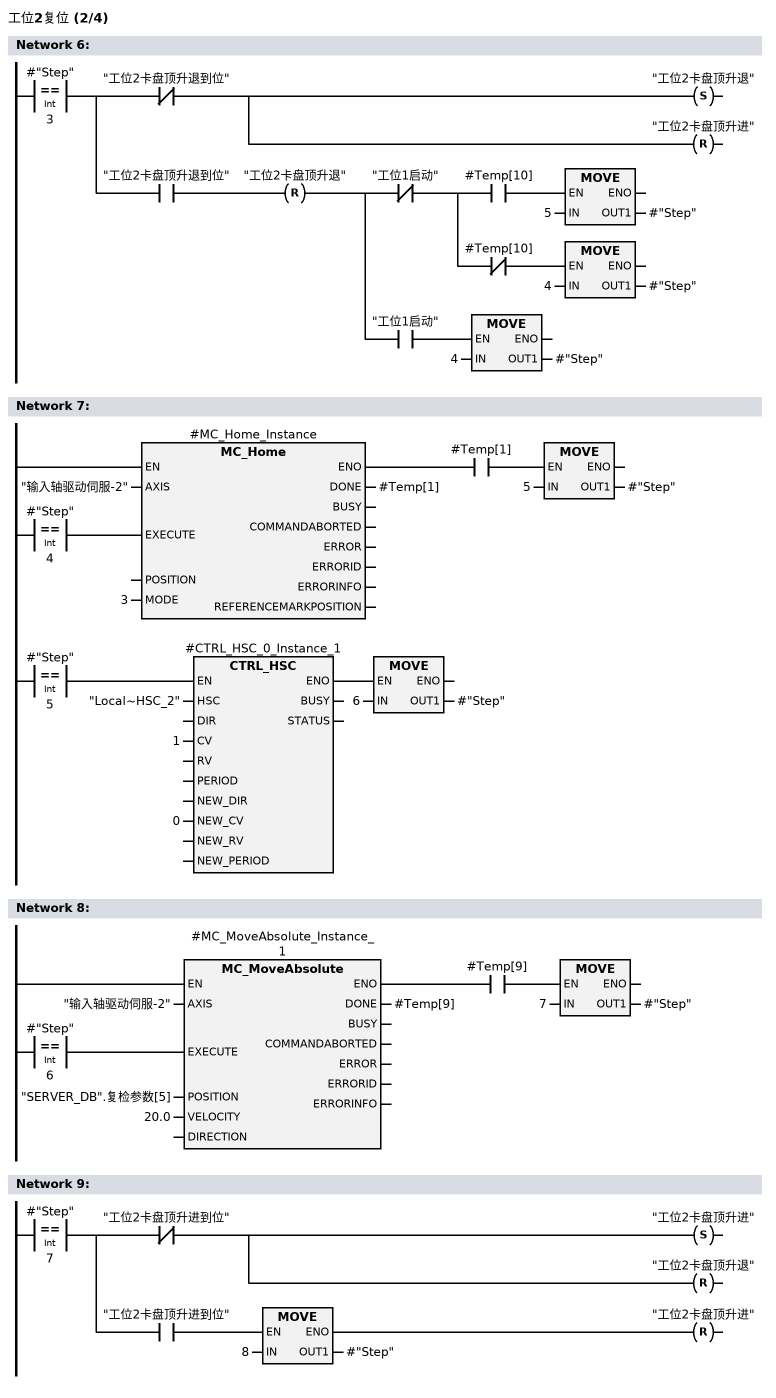
   RUNG wire#powerrail
      { S7_Templates := "SrcType := Int" } EQ_Contact(in1 := #"Step", in2 := 3)
      wire#w1
      I_Contact( "工位2卡盘顶升退到位" )
      wire#w2
      S_Coil( "工位2卡盘顶升退" )
   END_RUNG
   RUNG wire#w2
      R_Coil( "工位2卡盘顶升进" )
   END_RUNG
   RUNG wire#w1
      Contact( "工位2卡盘顶升退到位" )
      R_Coil( "工位2卡盘顶升退" )
      wire#w3
      I_Contact( "工位1启动" )
      wire#w4
      Contact( #Temp[10] )
      Move(in := 5, out1 => #"Step")
   END_RUNG
   RUNG wire#w4
      I_Contact( #Temp[10] )
      Move(in := 4, out1 => #"Step")
   END_RUNG
   RUNG wire#w3
      Contact( "工位1启动" )
      Move(in := 4, out1 => #"Step")
   END_RUNG
   // the same network as SCL:
   #_w1 := #"Step" = 3;
   IF #_w1 AND NOT "工位2卡盘顶升退到位" THEN
       "工位2卡盘顶升退" := TRUE;
       "工位2卡盘顶升进" := FALSE;
   END_IF;
   #_w2 := #_w1 AND "工位2卡盘顶升退到位";
   IF #_w2 THEN "工位2卡盘顶升退" := FALSE; END_IF;
   #_w3 := #_w2 AND NOT "工位1启动";
   IF #_w3 AND #Temp[10] THEN #"Step" := 5; END_IF;
   IF #_w3 AND NOT #Temp[10] THEN #"Step" := 4; END_IF;
   IF #_w2 AND "工位1启动" THEN #"Step" := 4; END_IF;
END_REGION

REGION Network 7
   // ENO of a box is taken as its EN; it also drops when the box reports an error
   #MC_Home_Instance(Axis := "输入轴驱动伺服-2", Execute := #"Step" = 4, Mode := 3, Done => #Temp[1]);   // MC_Home
   IF #Temp[1] THEN #"Step" := 5; END_IF;
   IF #"Step" = 5 THEN
       #CTRL_HSC_0_Instance_1(HSC := "Local~HSC_2", CV := 1, NEW_CV := 0);   // CTRL_HSC
       #"Step" := 6;
   END_IF;
END_REGION

REGION Network 8
   // ENO of a box is taken as its EN; it also drops when the box reports an error
   #MC_MoveAbsolute_Instance_1(Axis := "输入轴驱动伺服-2",   // MC_MoveAbsolute
                           Execute := #"Step" = 6,
                           Position := "SERVER_DB".复检参数[5],
                           Velocity := 20.0,
                           Done => #Temp[9]);
   IF #Temp[9] THEN #"Step" := 7; END_IF;
END_REGION

REGION Network 9
   RUNG wire#powerrail
      { S7_Templates := "SrcType := Int" } EQ_Contact(in1 := #"Step", in2 := 7)
      wire#w1
      I_Contact( "工位2卡盘顶升进到位" )
      wire#w2
      S_Coil( "工位2卡盘顶升进" )
   END_RUNG
   RUNG wire#w2
      R_Coil( "工位2卡盘顶升退" )
   END_RUNG
   RUNG wire#w1
      Contact( "工位2卡盘顶升进到位" )
      Move(in := 8, out1 => #"Step")
      R_Coil( "工位2卡盘顶升进" )
   END_RUNG
   // the same network as SCL:
   #_w1 := #"Step" = 7;
   IF #_w1 AND NOT "工位2卡盘顶升进到位" THEN
       "工位2卡盘顶升进" := TRUE;
       "工位2卡盘顶升退" := FALSE;
   END_IF;
   IF #_w1 AND "工位2卡盘顶升进到位" THEN
       #"Step" := 8;
       "工位2卡盘顶升进" := FALSE;
   END_IF;
END_REGION

REGION Network 10
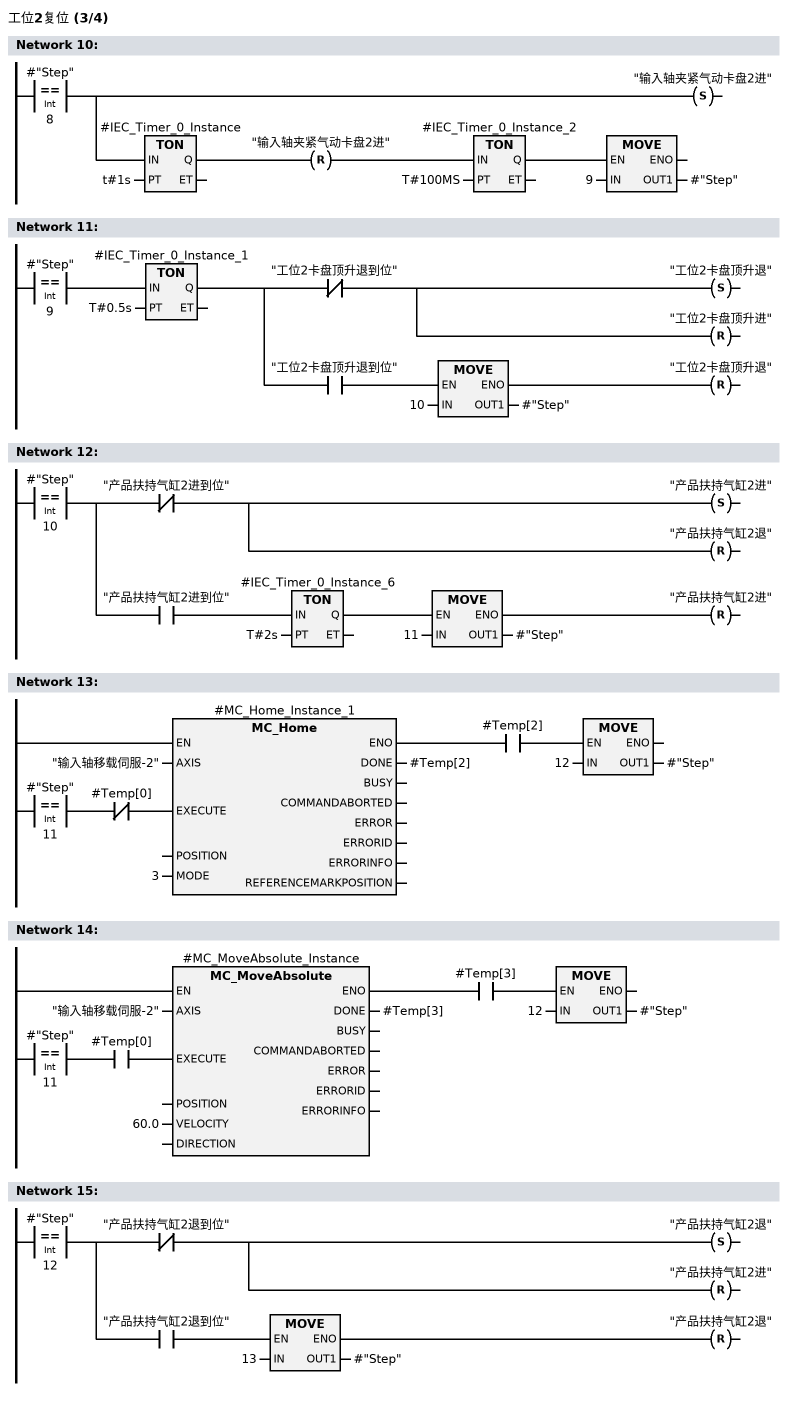
   #_w1 := #"Step" = 8;
   IF #_w1 THEN "输入轴夹紧气动卡盘2进" := TRUE; END_IF;
   #IEC_Timer_0_Instance(IN := #_w1, PT := t#1s);   // TON
   IF #IEC_Timer_0_Instance.Q THEN "输入轴夹紧气动卡盘2进" := FALSE; END_IF;
   #IEC_Timer_0_Instance_2(IN := #IEC_Timer_0_Instance.Q, PT := T#100MS);   // TON
   IF #IEC_Timer_0_Instance_2.Q THEN #"Step" := 9; END_IF;
END_REGION

REGION Network 11
   #IEC_Timer_0_Instance_1(IN := #"Step" = 9, PT := T#0.5s);   // TON
   IF #IEC_Timer_0_Instance_1.Q AND NOT "工位2卡盘顶升退到位" THEN
       "工位2卡盘顶升退" := TRUE;
       "工位2卡盘顶升进" := FALSE;
   END_IF;
   IF #IEC_Timer_0_Instance_1.Q AND "工位2卡盘顶升退到位" THEN
       #"Step" := 10;
       "工位2卡盘顶升退" := FALSE;
   END_IF;
END_REGION

REGION Network 12
   #_w1 := #"Step" = 10;
   IF #_w1 AND NOT "产品扶持气缸2进到位" THEN
       "产品扶持气缸2进" := TRUE;
       "产品扶持气缸2退" := FALSE;
   END_IF;
   #IEC_Timer_0_Instance_6(IN := #_w1 AND "产品扶持气缸2进到位", PT := T#2s);   // TON
   IF #IEC_Timer_0_Instance_6.Q THEN
       #"Step" := 11;
       "产品扶持气缸2进" := FALSE;
   END_IF;
END_REGION

REGION Network 13
   // ENO of a box is taken as its EN; it also drops when the box reports an error
   #MC_Home_Instance_1(Axis := "输入轴移载伺服-2",   // MC_Home
                       Execute := (#"Step" = 11) AND NOT #Temp[0],
                       Mode := 3,
                       Done => #Temp[2]);
   IF #Temp[2] THEN #"Step" := 12; END_IF;
END_REGION

REGION Network 14
   // ENO of a box is taken as its EN; it also drops when the box reports an error
   #MC_MoveAbsolute_Instance(Axis := "输入轴移载伺服-2",   // MC_MoveAbsolute
                           Execute := (#"Step" = 11) AND #Temp[0],
                           Velocity := 60.0,
                           Done => #Temp[3]);
   IF #Temp[3] THEN #"Step" := 12; END_IF;
END_REGION

REGION Network 15
   RUNG wire#powerrail
      { S7_Templates := "SrcType := Int" } EQ_Contact(in1 := #"Step", in2 := 12)
      wire#w1
      I_Contact( "产品扶持气缸2退到位" )
      wire#w2
      S_Coil( "产品扶持气缸2退" )
   END_RUNG
   RUNG wire#w2
      R_Coil( "产品扶持气缸2进" )
   END_RUNG
   RUNG wire#w1
      Contact( "产品扶持气缸2退到位" )
      Move(in := 13, out1 => #"Step")
      R_Coil( "产品扶持气缸2退" )
   END_RUNG
   // the same network as SCL:
   #_w1 := #"Step" = 12;
   IF #_w1 AND NOT "产品扶持气缸2退到位" THEN
       "产品扶持气缸2退" := TRUE;
       "产品扶持气缸2进" := FALSE;
   END_IF;
   IF #_w1 AND "产品扶持气缸2退到位" THEN
       #"Step" := 13;
       "产品扶持气缸2退" := FALSE;
   END_IF;
END_REGION

REGION Network 16
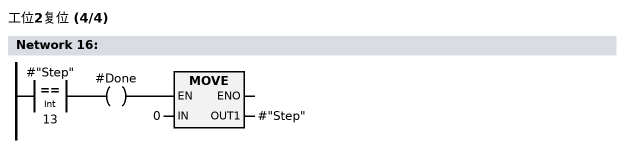
   RUNG wire#powerrail
      { S7_Templates := "SrcType := Int" } EQ_Contact(in1 := #"Step", in2 := 13)
      Coil( #Done )
      Move(in := 0, out1 => #"Step")
   END_RUNG
   // the same network as SCL:
   #Done := #"Step" = 13;
   IF #Done THEN #"Step" := 0; END_IF;
END_REGION
END_FUNCTION_BLOCK

FUNCTION_BLOCK "Auto1"   // FB9, LAD
{ S7_Optimized_Access := 'TRUE' }
VERSION : 0.1
   VAR
      Temp : Array[0..20] of Bool;
      newCV : DInt;
      输入轴移载下降夹紧_Instance : "工位1输入轴移载夹紧";
      复检_Instance : "工位1复检";
      复检_Instance_1 : "工位1复检";
      复检_Instance_2 : "工位1复检";
      复检_Instance_3 : "工位1复检";
      MC_Halt_Instance : MC_Halt;
      工位1复位_Instance : "工位1复位";
      复检_Instance_4 : "工位1复检";
      复检_Instance_5 : "工位1复检";
      IEC_Timer_0_Instance : TON_TIME;
      IEC_Timer_0_Instance_1 : TON_TIME;
      MC_MoveAbsolute_Instance : MC_MoveAbsolute;
      MC_MoveAbsolute_Instance_1 : MC_MoveAbsolute;
      MC_MoveAbsolute_Instance_2 : MC_MoveAbsolute;
      MC_MoveRelative_Instance : MC_MoveRelative;
      MC_MoveRelative_Instance_1 : MC_MoveRelative;
      MC_MoveRelative_Instance_2 : MC_MoveRelative;
      MC_MoveRelative_Instance_3 : MC_MoveRelative;
      MC_MoveRelative_Instance_4 : MC_MoveRelative;
      IEC_Timer_0_Instance_2 : TON_TIME;
      IEC_Timer_0_Instance_3 : TON_TIME;
   END_VAR
   VAR RETAIN
      IEC_Counter_0_Instance : CTU_INT;
   END_VAR
   VAR
      CTRL_HSC_0_Instance : CTRL_HSC;
      IEC_Timer_0_Instance_4 : TON_TIME;
      MC_MoveRelative_Instance_5 : MC_MoveRelative;
      工位1复检_Instance : "工位1复检";
      工位1复检_Instance_1 : "工位1复检";
      工位1复检_Instance_2 : "工位1复检";
   END_VAR
   VAR_TEMP   // added for the SCL form of the ladder/FBD networks
      _w1 : Bool;
      _w2 : Bool;
      _w3 : Bool;
   END_VAR
BEGIN

REGION Network 1
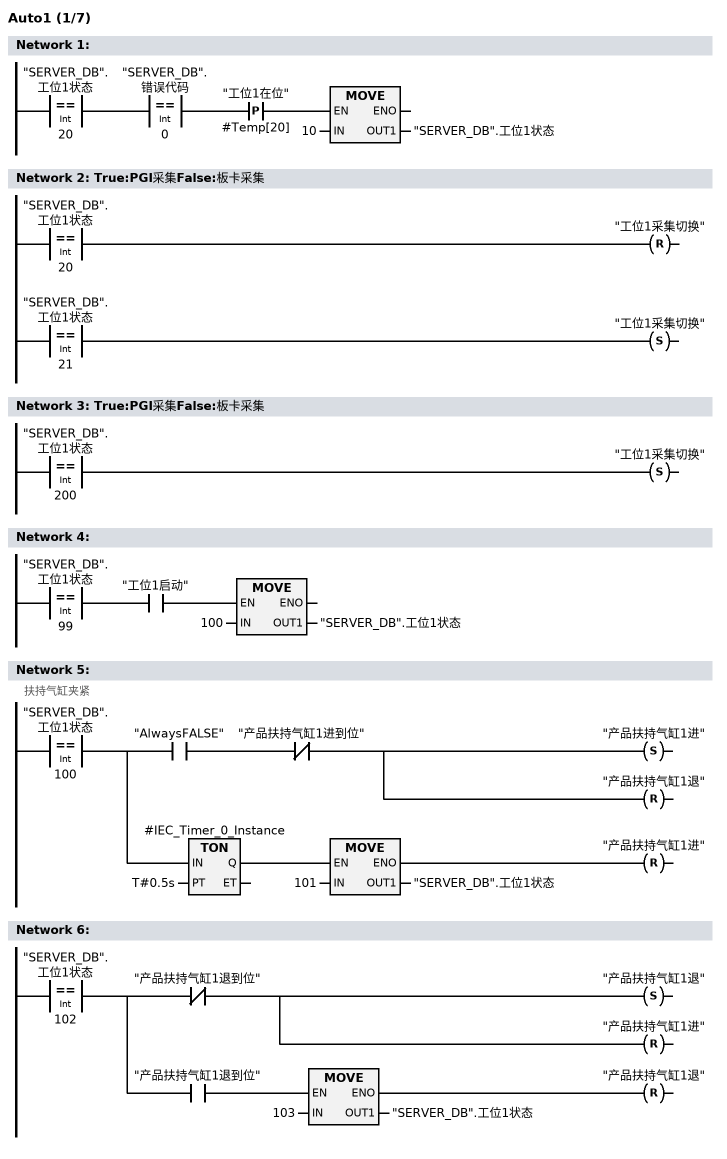
   RUNG wire#powerrail
      { S7_Templates := "SrcType := Int" } EQ_Contact(in1 := "SERVER_DB".工位1状态, in2 := 20)
      { S7_Templates := "SrcType := Int" } EQ_Contact(in1 := "SERVER_DB".错误代码, in2 := 0)
      P_Contact(operand := "工位1在位", bit := #Temp[20])
      Move(in := 10, out1 => "SERVER_DB".工位1状态)
   END_RUNG
   // the same network as SCL:
   #_w1 := ("SERVER_DB".工位1状态 = 20) AND ("SERVER_DB".错误代码 = 0) AND "工位1在位" AND NOT #Temp[20];   // rising edge of "工位1在位"
   #Temp[20] := "工位1在位";
   IF #_w1 THEN "SERVER_DB".工位1状态 := 10; END_IF;
END_REGION

REGION Network 2: True:PGI采集False:板卡采集
   RUNG wire#powerrail
      { S7_Templates := "SrcType := Int" } EQ_Contact(in1 := "SERVER_DB".工位1状态, in2 := 20)
      R_Coil( "工位1采集切换" )
   END_RUNG
   RUNG wire#powerrail
      { S7_Templates := "SrcType := Int" } EQ_Contact(in1 := "SERVER_DB".工位1状态, in2 := 21)
      S_Coil( "工位1采集切换" )
   END_RUNG
   // the same network as SCL:
   IF "SERVER_DB".工位1状态 = 20 THEN "工位1采集切换" := FALSE; END_IF;
   IF "SERVER_DB".工位1状态 = 21 THEN "工位1采集切换" := TRUE; END_IF;
END_REGION

REGION Network 3: True:PGI采集False:板卡采集
   RUNG wire#powerrail
      { S7_Templates := "SrcType := Int" } EQ_Contact(in1 := "SERVER_DB".工位1状态, in2 := 200)
      S_Coil( "工位1采集切换" )
   END_RUNG
   // the same network as SCL:
   IF "SERVER_DB".工位1状态 = 200 THEN "工位1采集切换" := TRUE; END_IF;
END_REGION

REGION Network 4
   RUNG wire#powerrail
      { S7_Templates := "SrcType := Int" } EQ_Contact(in1 := "SERVER_DB".工位1状态, in2 := 99)
      Contact( "工位1启动" )
      Move(in := 100, out1 => "SERVER_DB".工位1状态)
   END_RUNG
   // the same network as SCL:
   IF ("SERVER_DB".工位1状态 = 99) AND "工位1启动" THEN "SERVER_DB".工位1状态 := 100; END_IF;
END_REGION

REGION Network 5
   // 扶持气缸夹紧
   #_w1 := "SERVER_DB".工位1状态 = 100;
   IF #_w1 AND "AlwaysFALSE" AND NOT "产品扶持气缸1进到位" THEN
       "产品扶持气缸1进" := TRUE;
       "产品扶持气缸1退" := FALSE;
   END_IF;
   #IEC_Timer_0_Instance(IN := #_w1, PT := T#0.5s);   // TON
   IF #IEC_Timer_0_Instance.Q THEN
       "SERVER_DB".工位1状态 := 101;
       "产品扶持气缸1进" := FALSE;
   END_IF;
END_REGION

REGION Network 6
   RUNG wire#powerrail
      { S7_Templates := "SrcType := Int" } EQ_Contact(in1 := "SERVER_DB".工位1状态, in2 := 102)
      wire#w1
      I_Contact( "产品扶持气缸1退到位" )
      wire#w2
      S_Coil( "产品扶持气缸1退" )
   END_RUNG
   RUNG wire#w2
      R_Coil( "产品扶持气缸1进" )
   END_RUNG
   RUNG wire#w1
      Contact( "产品扶持气缸1退到位" )
      Move(in := 103, out1 => "SERVER_DB".工位1状态)
      R_Coil( "产品扶持气缸1退" )
   END_RUNG
   // the same network as SCL:
   #_w1 := "SERVER_DB".工位1状态 = 102;
   IF #_w1 AND NOT "产品扶持气缸1退到位" THEN
       "产品扶持气缸1退" := TRUE;
       "产品扶持气缸1进" := FALSE;
   END_IF;
   IF #_w1 AND "产品扶持气缸1退到位" THEN
       "SERVER_DB".工位1状态 := 103;
       "产品扶持气缸1退" := FALSE;
   END_IF;
END_REGION

REGION Network 7
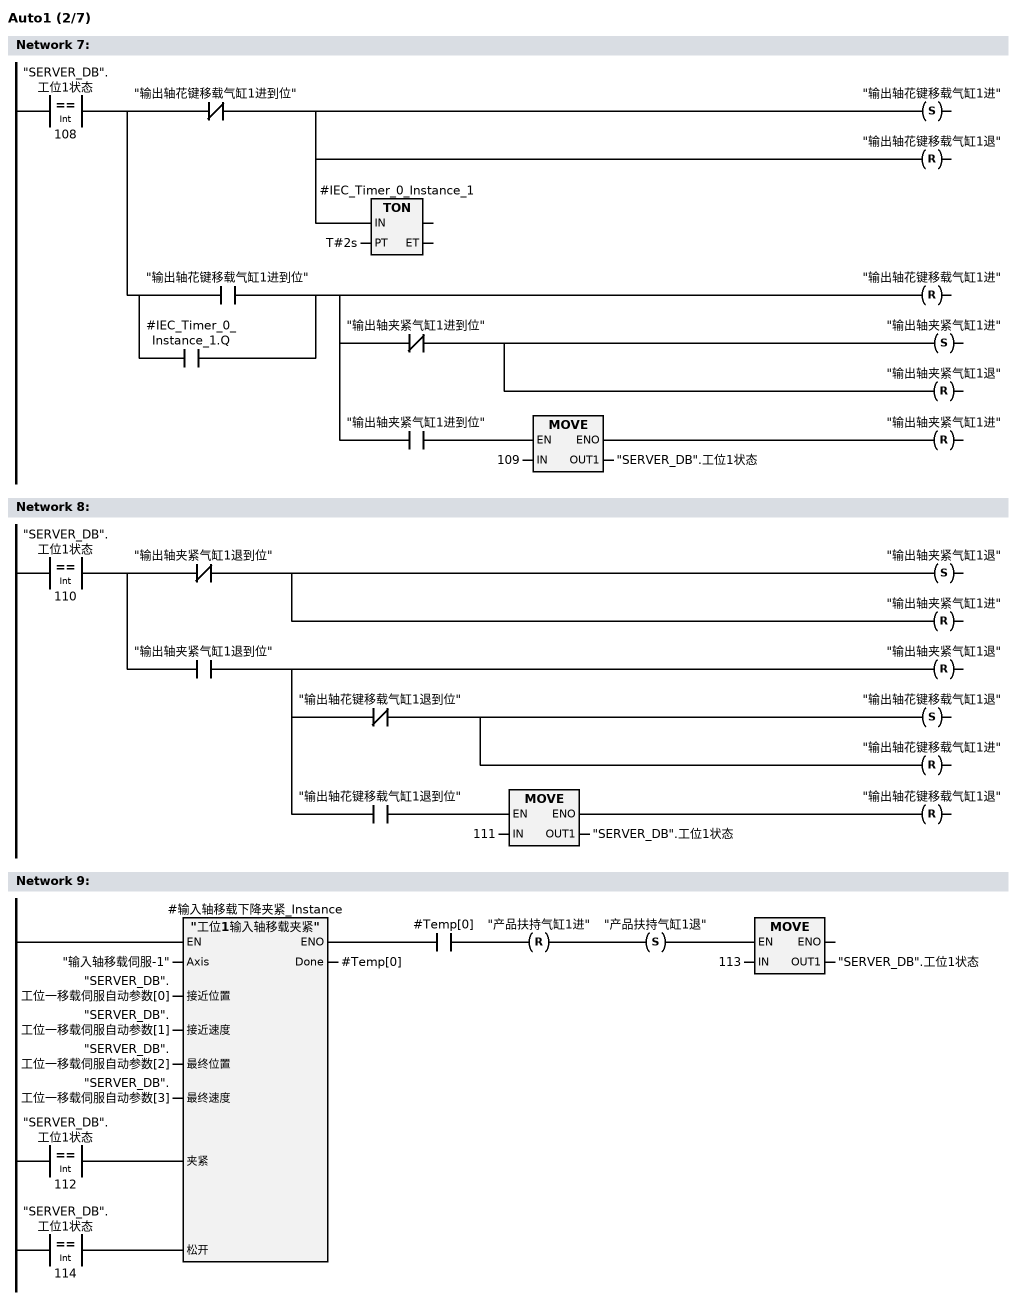
   #_w1 := "SERVER_DB".工位1状态 = 108;
   #_w2 := #_w1 AND NOT "输出轴花键移载气缸1进到位";
   IF #_w2 THEN
       "输出轴花键移载气缸1进" := TRUE;
       "输出轴花键移载气缸1退" := FALSE;
   END_IF;
   #IEC_Timer_0_Instance_1(IN := #_w2, PT := T#2s);   // TON
   #_w3 := #_w1 AND ("输出轴花键移载气缸1进到位" OR #IEC_Timer_0_Instance_1.Q);
   IF #_w3 THEN "输出轴花键移载气缸1进" := FALSE; END_IF;
   IF #_w3 AND NOT "输出轴夹紧气缸1进到位" THEN
       "输出轴夹紧气缸1进" := TRUE;
       "输出轴夹紧气缸1退" := FALSE;
   END_IF;
   IF #_w3 AND "输出轴夹紧气缸1进到位" THEN
       "SERVER_DB".工位1状态 := 109;
       "输出轴夹紧气缸1进" := FALSE;
   END_IF;
END_REGION

REGION Network 8
   RUNG wire#powerrail
      { S7_Templates := "SrcType := Int" } EQ_Contact(in1 := "SERVER_DB".工位1状态, in2 := 110)
      wire#w1
      I_Contact( "输出轴夹紧气缸1退到位" )
      wire#w2
      S_Coil( "输出轴夹紧气缸1退" )
   END_RUNG
   RUNG wire#w2
      R_Coil( "输出轴夹紧气缸1进" )
   END_RUNG
   RUNG wire#w1
      Contact( "输出轴夹紧气缸1退到位" )
      wire#w3
      R_Coil( "输出轴夹紧气缸1退" )
   END_RUNG
   RUNG wire#w3
      I_Contact( "输出轴花键移载气缸1退到位" )
      wire#w4
      S_Coil( "输出轴花键移载气缸1退" )
   END_RUNG
   RUNG wire#w4
      R_Coil( "输出轴花键移载气缸1进" )
   END_RUNG
   RUNG wire#w3
      Contact( "输出轴花键移载气缸1退到位" )
      Move(in := 111, out1 => "SERVER_DB".工位1状态)
      R_Coil( "输出轴花键移载气缸1退" )
   END_RUNG
   // the same network as SCL:
   #_w1 := "SERVER_DB".工位1状态 = 110;
   IF #_w1 AND NOT "输出轴夹紧气缸1退到位" THEN
       "输出轴夹紧气缸1退" := TRUE;
       "输出轴夹紧气缸1进" := FALSE;
   END_IF;
   #_w2 := #_w1 AND "输出轴夹紧气缸1退到位";
   IF #_w2 THEN "输出轴夹紧气缸1退" := FALSE; END_IF;
   IF #_w2 AND NOT "输出轴花键移载气缸1退到位" THEN
       "输出轴花键移载气缸1退" := TRUE;
       "输出轴花键移载气缸1进" := FALSE;
   END_IF;
   IF #_w2 AND "输出轴花键移载气缸1退到位" THEN
       "SERVER_DB".工位1状态 := 111;
       "输出轴花键移载气缸1退" := FALSE;
   END_IF;
END_REGION

REGION Network 9
   RUNG wire#powerrail
      #输入轴移载下降夹紧_Instance(夹紧 := wire#w1, 松开 := wire#w2, Axis := "输入轴移载伺服-1", 接近位置 := "SERVER_DB".工位一移载伺服自动参数[0], 接近速度 := "SERVER_DB".工位一移载伺服自动参数[1], 最终位置 := "SERVER_DB".工位一移载伺服自动参数[2], 最终速度 := "SERVER_DB".工位一移载伺服自动参数[3], Done => #Temp[0])
      Contact( #Temp[0] )
      R_Coil( "产品扶持气缸1进" )
      S_Coil( "产品扶持气缸1退" )
      Move(in := 113, out1 => "SERVER_DB".工位1状态)
   END_RUNG
   RUNG wire#powerrail
      { S7_Templates := "SrcType := Int" } EQ_Contact(in1 := "SERVER_DB".工位1状态, in2 := 112)
   END_RUNG wire#w1
   RUNG wire#powerrail
      { S7_Templates := "SrcType := Int" } EQ_Contact(in1 := "SERVER_DB".工位1状态, in2 := 114)
   END_RUNG wire#w2
   // the same network as SCL:
   #输入轴移载下降夹紧_Instance(Axis := "输入轴移载伺服-1",   // "工位1输入轴移载夹紧"
                       接近位置 := "SERVER_DB".工位一移载伺服自动参数[0],
                       接近速度 := "SERVER_DB".工位一移载伺服自动参数[1],
                       最终位置 := "SERVER_DB".工位一移载伺服自动参数[2],
                       最终速度 := "SERVER_DB".工位一移载伺服自动参数[3],
                       夹紧 := "SERVER_DB".工位1状态 = 112,
                       松开 := "SERVER_DB".工位1状态 = 114,
                       Done => #Temp[0],
                       ENO => #_w1);
   IF #_w1 AND #Temp[0] THEN
       "产品扶持气缸1进" := FALSE;
       "产品扶持气缸1退" := TRUE;
       "SERVER_DB".工位1状态 := 113;
   END_IF;
END_REGION

REGION Network 10: True:板卡供电False:PGI供电
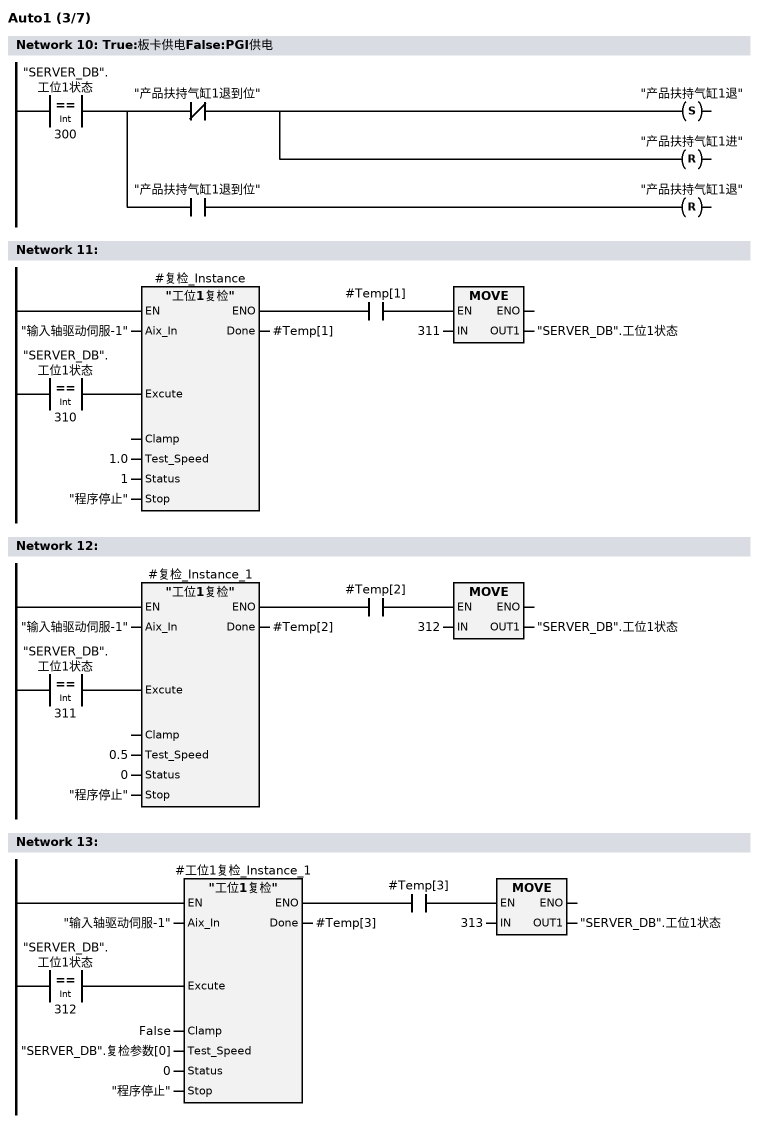
   RUNG wire#powerrail
      { S7_Templates := "SrcType := Int" } EQ_Contact(in1 := "SERVER_DB".工位1状态, in2 := 300)
      wire#w1
      I_Contact( "产品扶持气缸1退到位" )
      wire#w2
      S_Coil( "产品扶持气缸1退" )
   END_RUNG
   RUNG wire#w2
      R_Coil( "产品扶持气缸1进" )
   END_RUNG
   RUNG wire#w1
      Contact( "产品扶持气缸1退到位" )
      R_Coil( "产品扶持气缸1退" )
   END_RUNG
   // the same network as SCL:
   #_w1 := "SERVER_DB".工位1状态 = 300;
   IF #_w1 AND NOT "产品扶持气缸1退到位" THEN
       "产品扶持气缸1退" := TRUE;
       "产品扶持气缸1进" := FALSE;
   END_IF;
   IF #_w1 AND "产品扶持气缸1退到位" THEN "产品扶持气缸1退" := FALSE; END_IF;
END_REGION

REGION Network 11
   RUNG wire#powerrail
      #复检_Instance(Excute := wire#w1, Aix_In := "输入轴驱动伺服-1", Clamp :=, Test_Speed := 1.0, Status := 1, Stop := "程序停止", Done => #Temp[1])
      Contact( #Temp[1] )
      Move(in := 311, out1 => "SERVER_DB".工位1状态)
   END_RUNG
   RUNG wire#powerrail
      { S7_Templates := "SrcType := Int" } EQ_Contact(in1 := "SERVER_DB".工位1状态, in2 := 310)
   END_RUNG wire#w1
   // the same network as SCL:
   #复检_Instance(Aix_In := "输入轴驱动伺服-1",   // "工位1复检"
                Excute := "SERVER_DB".工位1状态 = 310,
                Test_Speed := 1.0,
                Status := 1,
                Stop := "程序停止",
                Done => #Temp[1],
                ENO => #_w1);
   IF #_w1 AND #Temp[1] THEN "SERVER_DB".工位1状态 := 311; END_IF;
END_REGION

REGION Network 12
   RUNG wire#powerrail
      #复检_Instance_1(Excute := wire#w1, Aix_In := "输入轴驱动伺服-1", Clamp :=, Test_Speed := 0.5, Status := 0, Stop := "程序停止", Done => #Temp[2])
      Contact( #Temp[2] )
      Move(in := 312, out1 => "SERVER_DB".工位1状态)
   END_RUNG
   RUNG wire#powerrail
      { S7_Templates := "SrcType := Int" } EQ_Contact(in1 := "SERVER_DB".工位1状态, in2 := 311)
   END_RUNG wire#w1
   // the same network as SCL:
   #复检_Instance_1(Aix_In := "输入轴驱动伺服-1",   // "工位1复检"
                  Excute := "SERVER_DB".工位1状态 = 311,
                  Test_Speed := 0.5,
                  Status := 0,
                  Stop := "程序停止",
                  Done => #Temp[2],
                  ENO => #_w1);
   IF #_w1 AND #Temp[2] THEN "SERVER_DB".工位1状态 := 312; END_IF;
END_REGION

REGION Network 13
   RUNG wire#powerrail
      #工位1复检_Instance_1(Excute := wire#w1, Aix_In := "输入轴驱动伺服-1", Clamp := False, Test_Speed := "SERVER_DB".复检参数[0], Status := 0, Stop := "程序停止", Done => #Temp[3])
      Contact( #Temp[3] )
      Move(in := 313, out1 => "SERVER_DB".工位1状态)
   END_RUNG
   RUNG wire#powerrail
      { S7_Templates := "SrcType := Int" } EQ_Contact(in1 := "SERVER_DB".工位1状态, in2 := 312)
   END_RUNG wire#w1
   // the same network as SCL:
   #工位1复检_Instance_1(Aix_In := "输入轴驱动伺服-1",   // "工位1复检"
                     Excute := "SERVER_DB".工位1状态 = 312,
                     Clamp := False,
                     Test_Speed := "SERVER_DB".复检参数[0],
                     Status := 0,
                     Stop := "程序停止",
                     Done => #Temp[3],
                     ENO => #_w1);
   IF #_w1 AND #Temp[3] THEN "SERVER_DB".工位1状态 := 313; END_IF;
END_REGION

REGION Network 14
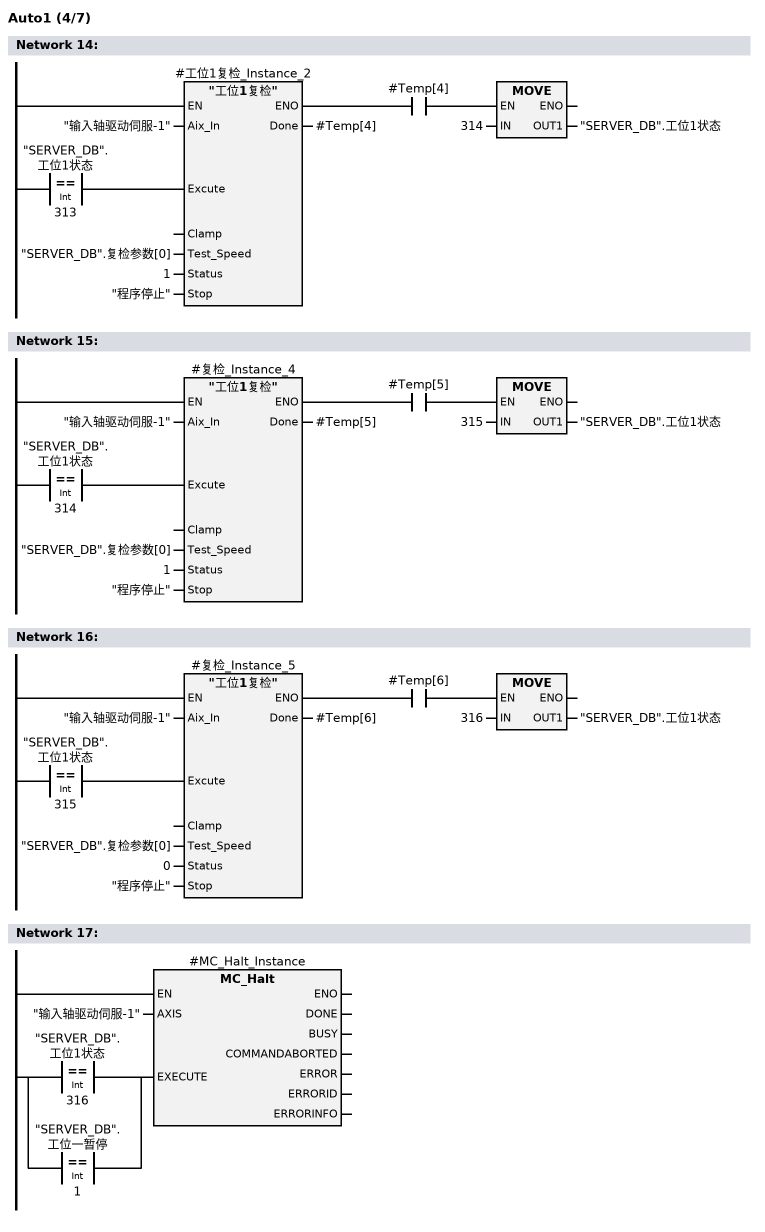
   RUNG wire#powerrail
      #工位1复检_Instance_2(Excute := wire#w1, Aix_In := "输入轴驱动伺服-1", Clamp :=, Test_Speed := "SERVER_DB".复检参数[0], Status := 1, Stop := "程序停止", Done => #Temp[4])
      Contact( #Temp[4] )
      Move(in := 314, out1 => "SERVER_DB".工位1状态)
   END_RUNG
   RUNG wire#powerrail
      { S7_Templates := "SrcType := Int" } EQ_Contact(in1 := "SERVER_DB".工位1状态, in2 := 313)
   END_RUNG wire#w1
   // the same network as SCL:
   #工位1复检_Instance_2(Aix_In := "输入轴驱动伺服-1",   // "工位1复检"
                     Excute := "SERVER_DB".工位1状态 = 313,
                     Test_Speed := "SERVER_DB".复检参数[0],
                     Status := 1,
                     Stop := "程序停止",
                     Done => #Temp[4],
                     ENO => #_w1);
   IF #_w1 AND #Temp[4] THEN "SERVER_DB".工位1状态 := 314; END_IF;
END_REGION

REGION Network 15
   RUNG wire#powerrail
      #复检_Instance_4(Excute := wire#w1, Aix_In := "输入轴驱动伺服-1", Clamp :=, Test_Speed := "SERVER_DB".复检参数[0], Status := 1, Stop := "程序停止", Done => #Temp[5])
      Contact( #Temp[5] )
      Move(in := 315, out1 => "SERVER_DB".工位1状态)
   END_RUNG
   RUNG wire#powerrail
      { S7_Templates := "SrcType := Int" } EQ_Contact(in1 := "SERVER_DB".工位1状态, in2 := 314)
   END_RUNG wire#w1
   // the same network as SCL:
   #复检_Instance_4(Aix_In := "输入轴驱动伺服-1",   // "工位1复检"
                  Excute := "SERVER_DB".工位1状态 = 314,
                  Test_Speed := "SERVER_DB".复检参数[0],
                  Status := 1,
                  Stop := "程序停止",
                  Done => #Temp[5],
                  ENO => #_w1);
   IF #_w1 AND #Temp[5] THEN "SERVER_DB".工位1状态 := 315; END_IF;
END_REGION

REGION Network 16
   RUNG wire#powerrail
      #复检_Instance_5(Excute := wire#w1, Aix_In := "输入轴驱动伺服-1", Clamp :=, Test_Speed := "SERVER_DB".复检参数[0], Status := 0, Stop := "程序停止", Done => #Temp[6])
      Contact( #Temp[6] )
      Move(in := 316, out1 => "SERVER_DB".工位1状态)
   END_RUNG
   RUNG wire#powerrail
      { S7_Templates := "SrcType := Int" } EQ_Contact(in1 := "SERVER_DB".工位1状态, in2 := 315)
   END_RUNG wire#w1
   // the same network as SCL:
   #复检_Instance_5(Aix_In := "输入轴驱动伺服-1",   // "工位1复检"
                  Excute := "SERVER_DB".工位1状态 = 315,
                  Test_Speed := "SERVER_DB".复检参数[0],
                  Status := 0,
                  Stop := "程序停止",
                  Done => #Temp[6],
                  ENO => #_w1);
   IF #_w1 AND #Temp[6] THEN "SERVER_DB".工位1状态 := 316; END_IF;
END_REGION

REGION Network 17
   #MC_Halt_Instance(Axis := "输入轴驱动伺服-1", Execute := ("SERVER_DB".工位1状态 = 316) OR ("SERVER_DB".工位一暂停 = 1));   // MC_Halt
END_REGION

REGION Network 18
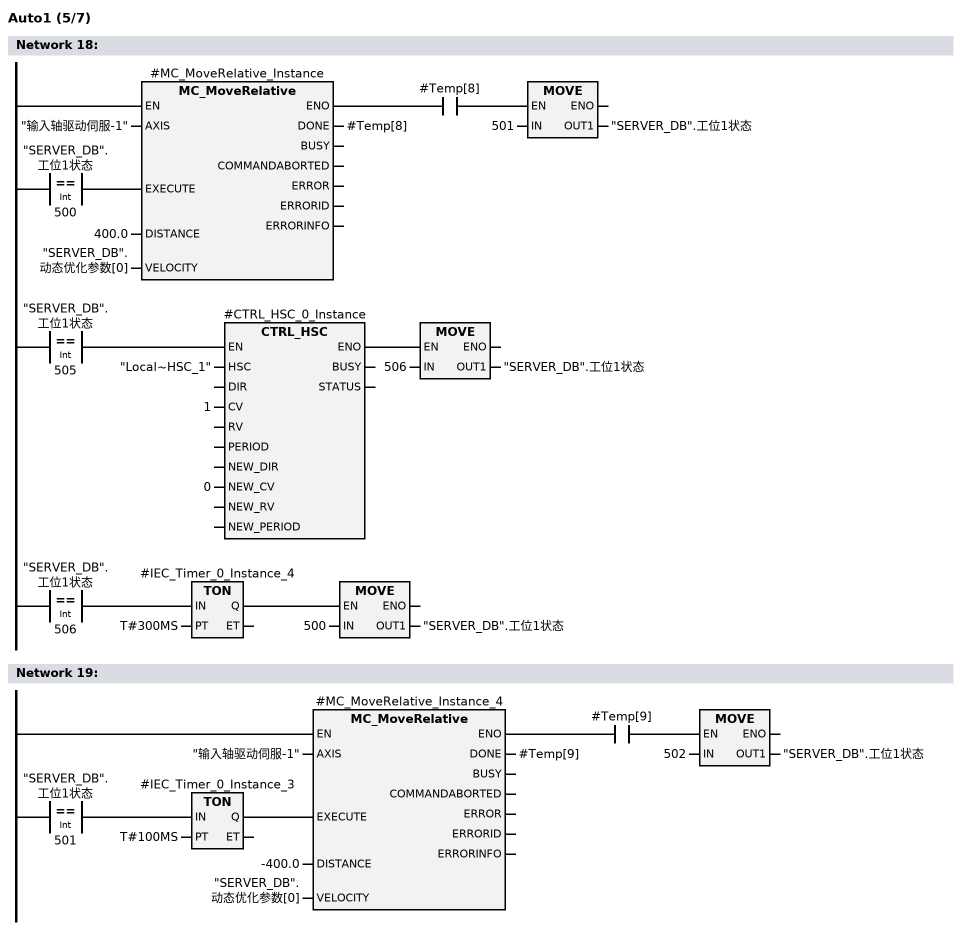
   // ENO of a box is taken as its EN; it also drops when the box reports an error
   #MC_MoveRelative_Instance(Axis := "输入轴驱动伺服-1",   // MC_MoveRelative
                           Execute := "SERVER_DB".工位1状态 = 500,
                           Distance := 400.0,
                           Velocity := "SERVER_DB".动态优化参数[0],
                           Done => #Temp[8]);
   IF #Temp[8] THEN "SERVER_DB".工位1状态 := 501; END_IF;
   #_w1 := "SERVER_DB".工位1状态 = 505;
   IF #_w1 THEN
       #CTRL_HSC_0_Instance(HSC := "Local~HSC_1", CV := 1, NEW_CV := 0);   // CTRL_HSC
       "SERVER_DB".工位1状态 := 506;
   END_IF;
   #IEC_Timer_0_Instance_4(IN := "SERVER_DB".工位1状态 = 506, PT := T#300MS);   // TON
   IF #IEC_Timer_0_Instance_4.Q THEN "SERVER_DB".工位1状态 := 500; END_IF;
END_REGION

REGION Network 19
   // ENO of a box is taken as its EN; it also drops when the box reports an error
   #IEC_Timer_0_Instance_3(IN := "SERVER_DB".工位1状态 = 501, PT := T#100MS);   // TON
   #MC_MoveRelative_Instance_4(Axis := "输入轴驱动伺服-1",   // MC_MoveRelative
                           Execute := #IEC_Timer_0_Instance_3.Q,
                           Distance := -400.0,
                           Velocity := "SERVER_DB".动态优化参数[0],
                           Done => #Temp[9]);
   IF #Temp[9] THEN "SERVER_DB".工位1状态 := 502; END_IF;
END_REGION

REGION Network 20
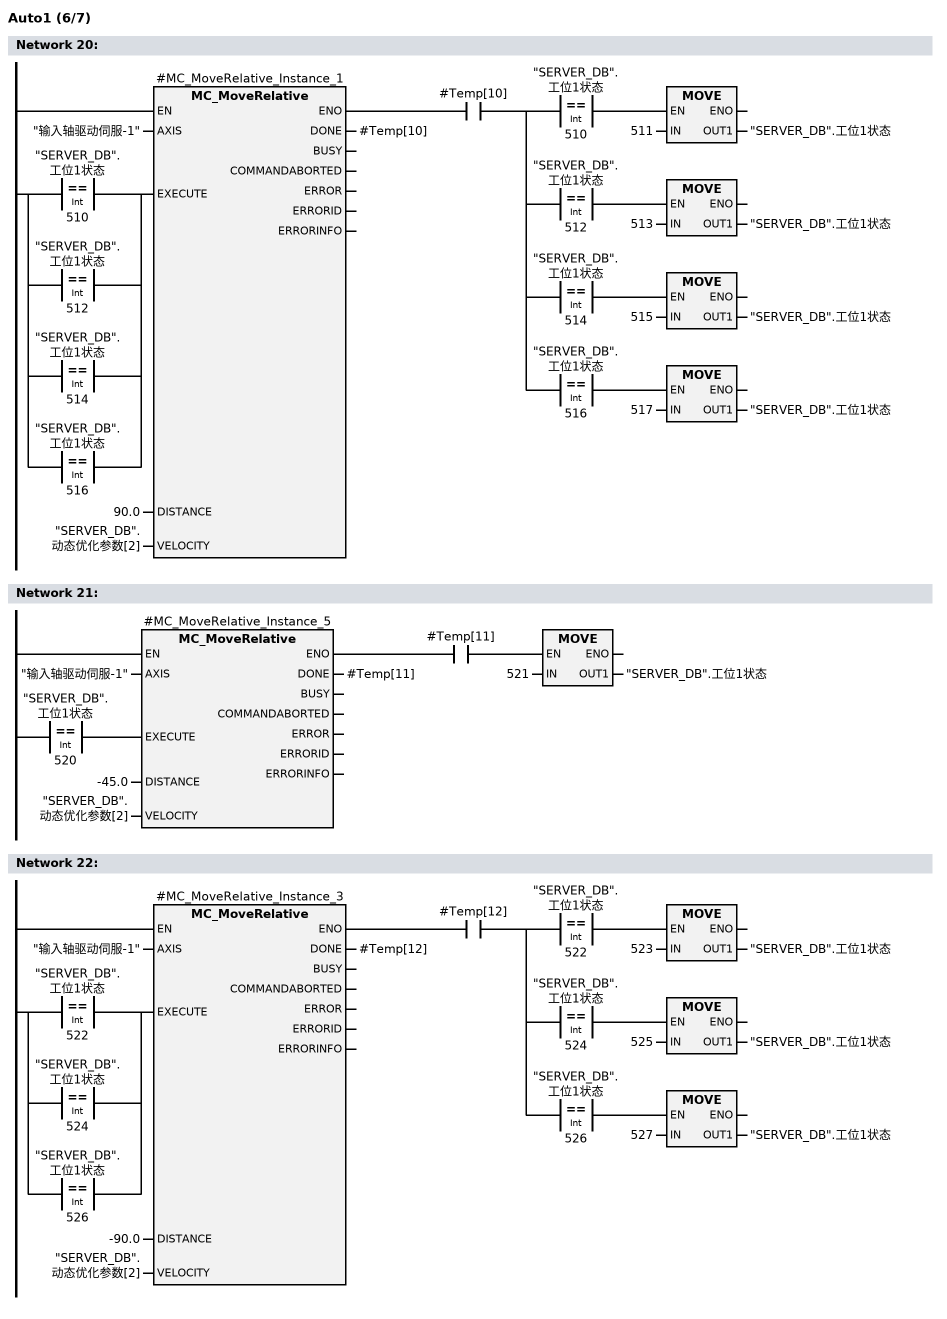
   // ENO of a box is taken as its EN; it also drops when the box reports an error
   #MC_MoveRelative_Instance_1(Axis := "输入轴驱动伺服-1",   // MC_MoveRelative
                           Execute := ("SERVER_DB".工位1状态 = 510) OR ("SERVER_DB".工位1状态 = 512) OR ("SERVER_DB".工位1状态 = 514) OR ("SERVER_DB".工位1状态 = 516),
                           Distance := 90.0,
                           Velocity := "SERVER_DB".动态优化参数[2],
                           Done => #Temp[10]);
   IF #Temp[10] AND ("SERVER_DB".工位1状态 = 510) THEN "SERVER_DB".工位1状态 := 511; END_IF;
   IF #Temp[10] AND ("SERVER_DB".工位1状态 = 512) THEN "SERVER_DB".工位1状态 := 513; END_IF;
   IF #Temp[10] AND ("SERVER_DB".工位1状态 = 514) THEN "SERVER_DB".工位1状态 := 515; END_IF;
   IF #Temp[10] AND ("SERVER_DB".工位1状态 = 516) THEN "SERVER_DB".工位1状态 := 517; END_IF;
END_REGION

REGION Network 21
   // ENO of a box is taken as its EN; it also drops when the box reports an error
   #MC_MoveRelative_Instance_5(Axis := "输入轴驱动伺服-1",   // MC_MoveRelative
                           Execute := "SERVER_DB".工位1状态 = 520,
                           Distance := -45.0,
                           Velocity := "SERVER_DB".动态优化参数[2],
                           Done => #Temp[11]);
   IF #Temp[11] THEN "SERVER_DB".工位1状态 := 521; END_IF;
END_REGION

REGION Network 22
   // ENO of a box is taken as its EN; it also drops when the box reports an error
   #MC_MoveRelative_Instance_3(Axis := "输入轴驱动伺服-1",   // MC_MoveRelative
                           Execute := ("SERVER_DB".工位1状态 = 522) OR ("SERVER_DB".工位1状态 = 524) OR ("SERVER_DB".工位1状态 = 526),
                           Distance := -90.0,
                           Velocity := "SERVER_DB".动态优化参数[2],
                           Done => #Temp[12]);
   IF #Temp[12] AND ("SERVER_DB".工位1状态 = 522) THEN "SERVER_DB".工位1状态 := 523; END_IF;
   IF #Temp[12] AND ("SERVER_DB".工位1状态 = 524) THEN "SERVER_DB".工位1状态 := 525; END_IF;
   IF #Temp[12] AND ("SERVER_DB".工位1状态 = 526) THEN "SERVER_DB".工位1状态 := 527; END_IF;
END_REGION

REGION Network 23
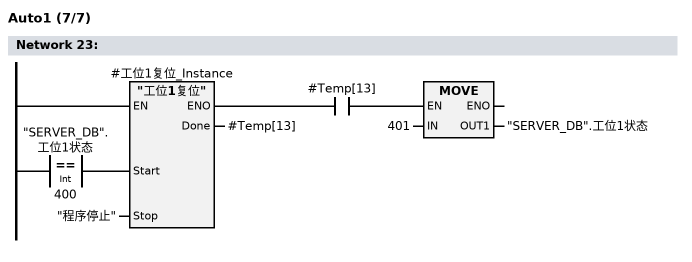
   RUNG wire#powerrail
      #工位1复位_Instance(Start := wire#w1, Stop := "程序停止", Done => #Temp[13])
      Contact( #Temp[13] )
      Move(in := 401, out1 => "SERVER_DB".工位1状态)
   END_RUNG
   RUNG wire#powerrail
      { S7_Templates := "SrcType := Int" } EQ_Contact(in1 := "SERVER_DB".工位1状态, in2 := 400)
   END_RUNG wire#w1
   // the same network as SCL:
   #工位1复位_Instance(Start := "SERVER_DB".工位1状态 = 400, Stop := "程序停止", Done => #Temp[13], ENO => #_w1);   // "工位1复位"
   IF #_w1 AND #Temp[13] THEN "SERVER_DB".工位1状态 := 401; END_IF;
END_REGION
END_FUNCTION_BLOCK

FUNCTION_BLOCK "工位1输入轴二次夹紧"   // FB10, LAD
{ S7_Optimized_Access := 'TRUE' }
VERSION : 0.1
   VAR_INPUT
      Axis : TO_PositioningAxis;
      Start : Bool;
      夹紧位置 : Real;
   END_VAR
   VAR_OUTPUT
      Done : Bool;
   END_VAR
   VAR
      "Step" : Int;
      Temp : Array[0..3] of Bool;
      MC_MoveAbsolute_Instance : MC_MoveAbsolute;
      IEC_Timer_0_Instance : TON_TIME;
      IEC_Timer_0_Instance_1 : TON_TIME;
   END_VAR
   VAR_TEMP   // added for the SCL form of the ladder/FBD networks
      _w1 : Bool;
   END_VAR
BEGIN

REGION Network 1
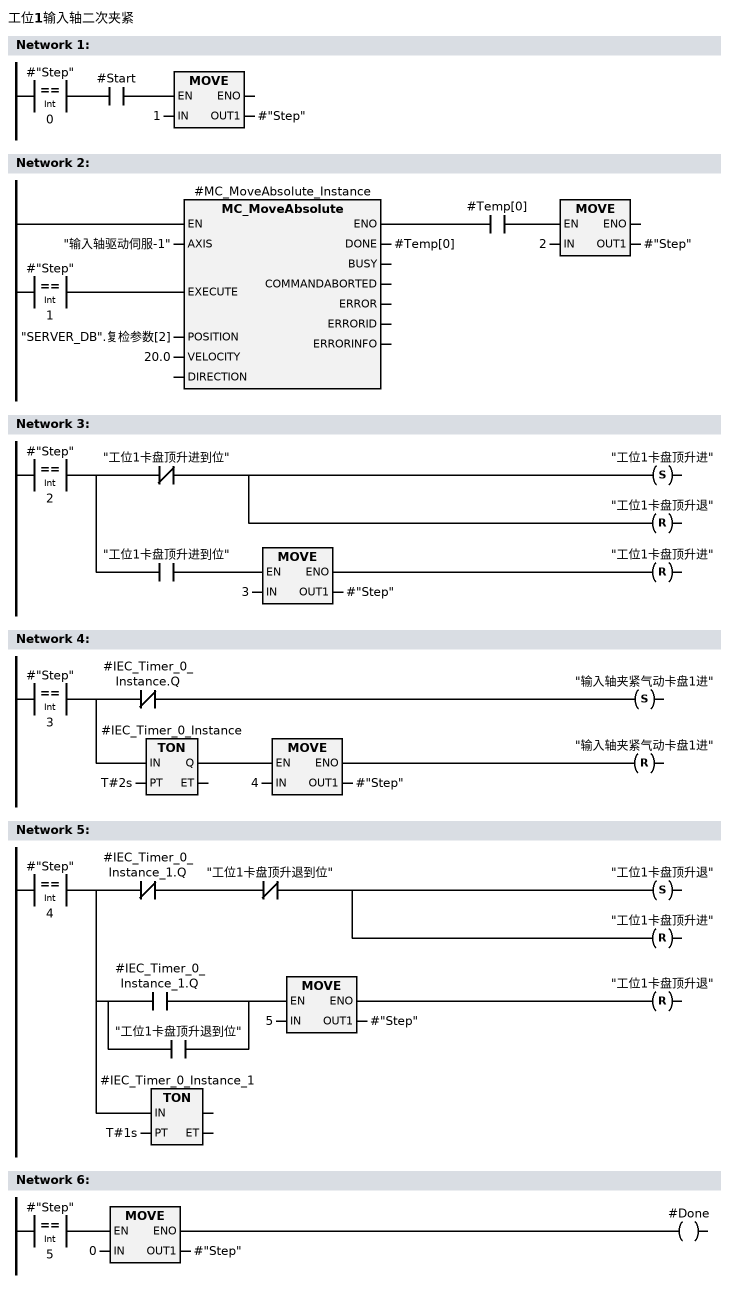
   RUNG wire#powerrail
      { S7_Templates := "SrcType := Int" } EQ_Contact(in1 := #"Step", in2 := 0)
      Contact( #Start )
      Move(in := 1, out1 => #"Step")
   END_RUNG
   // the same network as SCL:
   IF (#"Step" = 0) AND #Start THEN #"Step" := 1; END_IF;
END_REGION

REGION Network 2
   // ENO of a box is taken as its EN; it also drops when the box reports an error
   #MC_MoveAbsolute_Instance(Axis := "输入轴驱动伺服-1",   // MC_MoveAbsolute
                           Execute := #"Step" = 1,
                           Position := "SERVER_DB".复检参数[2],
                           Velocity := 20.0,
                           Done => #Temp[0]);
   IF #Temp[0] THEN #"Step" := 2; END_IF;
END_REGION

REGION Network 3
   RUNG wire#powerrail
      { S7_Templates := "SrcType := Int" } EQ_Contact(in1 := #"Step", in2 := 2)
      wire#w1
      I_Contact( "工位1卡盘顶升进到位" )
      wire#w2
      S_Coil( "工位1卡盘顶升进" )
   END_RUNG
   RUNG wire#w2
      R_Coil( "工位1卡盘顶升退" )
   END_RUNG
   RUNG wire#w1
      Contact( "工位1卡盘顶升进到位" )
      Move(in := 3, out1 => #"Step")
      R_Coil( "工位1卡盘顶升进" )
   END_RUNG
   // the same network as SCL:
   #_w1 := #"Step" = 2;
   IF #_w1 AND NOT "工位1卡盘顶升进到位" THEN
       "工位1卡盘顶升进" := TRUE;
       "工位1卡盘顶升退" := FALSE;
   END_IF;
   IF #_w1 AND "工位1卡盘顶升进到位" THEN
       #"Step" := 3;
       "工位1卡盘顶升进" := FALSE;
   END_IF;
END_REGION

REGION Network 4
   #_w1 := #"Step" = 3;
   IF #_w1 AND NOT #IEC_Timer_0_Instance.Q THEN "输入轴夹紧气动卡盘1进" := TRUE; END_IF;
   #IEC_Timer_0_Instance(IN := #_w1, PT := T#2s);   // TON
   IF #IEC_Timer_0_Instance.Q THEN
       #"Step" := 4;
       "输入轴夹紧气动卡盘1进" := FALSE;
   END_IF;
END_REGION

REGION Network 5
   #_w1 := #"Step" = 4;
   IF #_w1 AND NOT #IEC_Timer_0_Instance_1.Q AND NOT "工位1卡盘顶升退到位" THEN
       "工位1卡盘顶升退" := TRUE;
       "工位1卡盘顶升进" := FALSE;
   END_IF;
   IF #_w1 AND (#IEC_Timer_0_Instance_1.Q OR "工位1卡盘顶升退到位") THEN
       #"Step" := 5;
       "工位1卡盘顶升退" := FALSE;
   END_IF;
   #IEC_Timer_0_Instance_1(IN := #_w1, PT := T#1s);   // TON
END_REGION

REGION Network 6
   RUNG wire#powerrail
      { S7_Templates := "SrcType := Int" } EQ_Contact(in1 := #"Step", in2 := 5)
      Move(in := 0, out1 => #"Step")
      Coil( #Done )
   END_RUNG
   // the same network as SCL:
   #_w1 := #"Step" = 5;
   IF #_w1 THEN #"Step" := 0; END_IF;
   #Done := #_w1;
END_REGION
END_FUNCTION_BLOCK

FUNCTION_BLOCK "工位1输入轴移载夹紧"   // FB11, LAD
{ S7_Optimized_Access := 'TRUE' }
VERSION : 0.1
   VAR_INPUT
      Axis : TO_PositioningAxis;
      接近位置 : Real;
      接近速度 : Real;
      最终位置 : Real;
      最终速度 : Real;
      夹紧 : Bool;
      松开 : Bool;
   END_VAR
   VAR_OUTPUT
      Done : Bool;
   END_VAR
   VAR
      "Step" : Int;
      Temp : Array[0..7] of Bool;
      MC_MoveAbsolute_Instance : MC_MoveAbsolute;
      MC_MoveAbsolute_Instance_1 : MC_MoveAbsolute;
      MC_MoveAbsolute_Instance_2 : MC_MoveAbsolute;
      IEC_Timer_0_Instance : TON_TIME;
      IEC_Timer_0_Instance_1 : TON_TIME;
      MC_MoveAbsolute_Instance_3 : MC_MoveAbsolute;
      MC_MoveAbsolute_Instance_4 : MC_MoveAbsolute;
      MC_MoveAbsolute_Instance_5 : MC_MoveAbsolute;
      IEC_Timer_0_Instance_2 : TON_TIME;
      IEC_Timer_0_Instance_3 : TON_TIME;
      IEC_Timer_0_Instance_4 : TON_TIME;
      MC_MoveRelative_Instance : MC_MoveRelative;
      MC_MoveRelative_Instance_1 : MC_MoveRelative;
   END_VAR
   VAR RETAIN
      IEC_Counter_0_Instance : CTU_INT;
   END_VAR
   VAR
      MC_MoveRelative_Instance_2 : MC_MoveRelative;
      MC_MoveRelative_Instance_3 : MC_MoveRelative;
      IEC_Timer_0_Instance_5 : TON_TIME;
   END_VAR
   VAR_TEMP   // added for the SCL form of the ladder/FBD networks
      _w1 : Bool;
   END_VAR
BEGIN

REGION Network 1
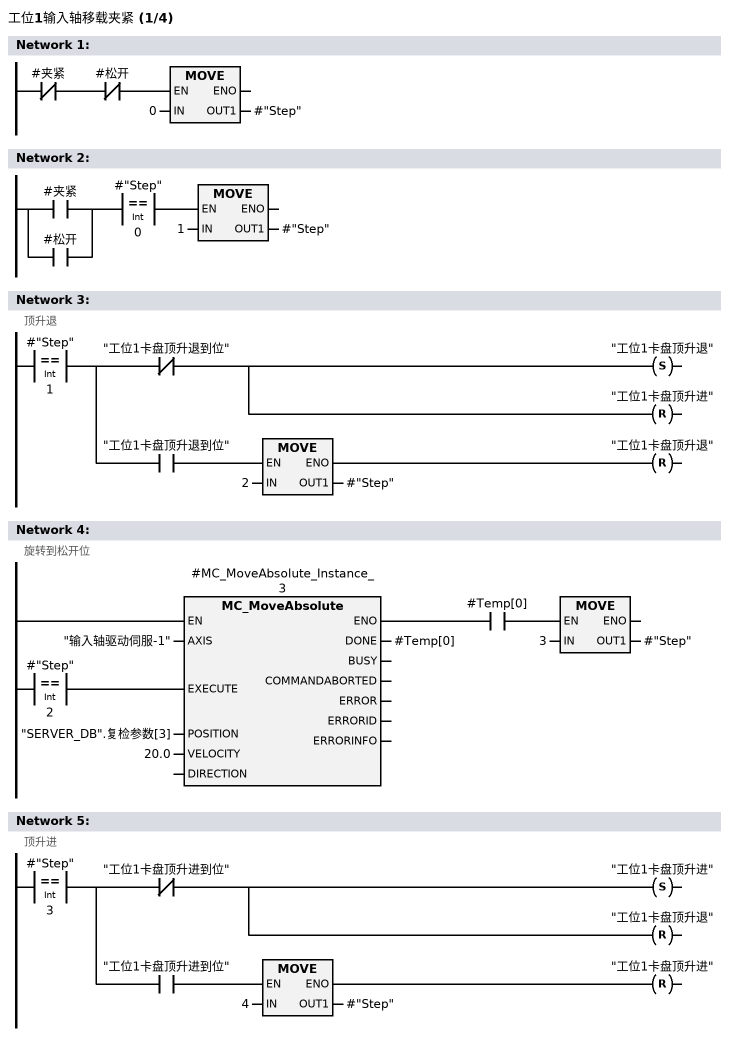
   RUNG wire#powerrail
      I_Contact( #夹紧 )
      I_Contact( #松开 )
      Move(in := 0, out1 => #"Step")
   END_RUNG
   // the same network as SCL:
   IF NOT #夹紧 AND NOT #松开 THEN #"Step" := 0; END_IF;
END_REGION

REGION Network 2
   RUNG wire#powerrail
      Contact( #夹紧 )
      wire#w1
      { S7_Templates := "SrcType := Int" } EQ_Contact(in1 := #"Step", in2 := 0)
      Move(in := 1, out1 => #"Step")
   END_RUNG
   RUNG wire#powerrail
      Contact( #松开 )
   END_RUNG wire#w1
   // the same network as SCL:
   IF (#夹紧 OR #松开) AND (#"Step" = 0) THEN #"Step" := 1; END_IF;
END_REGION

REGION Network 3
   // 顶升退
   RUNG wire#powerrail
      { S7_Templates := "SrcType := Int" } EQ_Contact(in1 := #"Step", in2 := 1)
      wire#w1
      I_Contact( "工位1卡盘顶升退到位" )
      wire#w2
      S_Coil( "工位1卡盘顶升退" )
   END_RUNG
   RUNG wire#w2
      R_Coil( "工位1卡盘顶升进" )
   END_RUNG
   RUNG wire#w1
      Contact( "工位1卡盘顶升退到位" )
      Move(in := 2, out1 => #"Step")
      R_Coil( "工位1卡盘顶升退" )
   END_RUNG
   // the same network as SCL:
   #_w1 := #"Step" = 1;
   IF #_w1 AND NOT "工位1卡盘顶升退到位" THEN
       "工位1卡盘顶升退" := TRUE;
       "工位1卡盘顶升进" := FALSE;
   END_IF;
   IF #_w1 AND "工位1卡盘顶升退到位" THEN
       #"Step" := 2;
       "工位1卡盘顶升退" := FALSE;
   END_IF;
END_REGION

REGION Network 4
   // 旋转到松开位
   // ENO of a box is taken as its EN; it also drops when the box reports an error
   #MC_MoveAbsolute_Instance_3(Axis := "输入轴驱动伺服-1",   // MC_MoveAbsolute
                           Execute := #"Step" = 2,
                           Position := "SERVER_DB".复检参数[3],
                           Velocity := 20.0,
                           Done => #Temp[0]);
   IF #Temp[0] THEN #"Step" := 3; END_IF;
END_REGION

REGION Network 5
   // 顶升进
   RUNG wire#powerrail
      { S7_Templates := "SrcType := Int" } EQ_Contact(in1 := #"Step", in2 := 3)
      wire#w1
      I_Contact( "工位1卡盘顶升进到位" )
      wire#w2
      S_Coil( "工位1卡盘顶升进" )
   END_RUNG
   RUNG wire#w2
      R_Coil( "工位1卡盘顶升退" )
   END_RUNG
   RUNG wire#w1
      Contact( "工位1卡盘顶升进到位" )
      Move(in := 4, out1 => #"Step")
      R_Coil( "工位1卡盘顶升进" )
   END_RUNG
   // the same network as SCL:
   #_w1 := #"Step" = 3;
   IF #_w1 AND NOT "工位1卡盘顶升进到位" THEN
       "工位1卡盘顶升进" := TRUE;
       "工位1卡盘顶升退" := FALSE;
   END_IF;
   IF #_w1 AND "工位1卡盘顶升进到位" THEN
       #"Step" := 4;
       "工位1卡盘顶升进" := FALSE;
   END_IF;
END_REGION

REGION Network 6
   // 卡盘松开
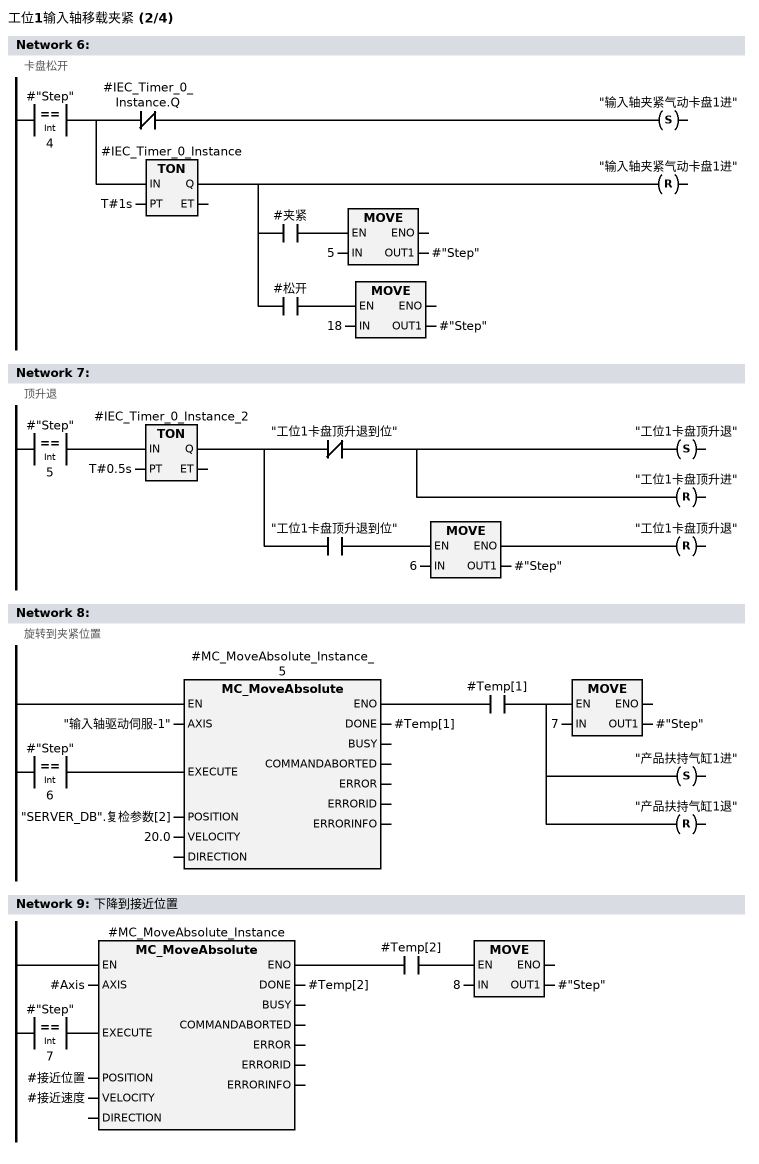
   #_w1 := #"Step" = 4;
   IF #_w1 AND NOT #IEC_Timer_0_Instance.Q THEN "输入轴夹紧气动卡盘1进" := TRUE; END_IF;
   #IEC_Timer_0_Instance(IN := #_w1, PT := T#1s);   // TON
   IF #IEC_Timer_0_Instance.Q THEN "输入轴夹紧气动卡盘1进" := FALSE; END_IF;
   IF #IEC_Timer_0_Instance.Q AND #夹紧 THEN #"Step" := 5; END_IF;
   IF #IEC_Timer_0_Instance.Q AND #松开 THEN #"Step" := 18; END_IF;
END_REGION

REGION Network 7
   // 顶升退
   #IEC_Timer_0_Instance_2(IN := #"Step" = 5, PT := T#0.5s);   // TON
   IF #IEC_Timer_0_Instance_2.Q AND NOT "工位1卡盘顶升退到位" THEN
       "工位1卡盘顶升退" := TRUE;
       "工位1卡盘顶升进" := FALSE;
   END_IF;
   IF #IEC_Timer_0_Instance_2.Q AND "工位1卡盘顶升退到位" THEN
       #"Step" := 6;
       "工位1卡盘顶升退" := FALSE;
   END_IF;
END_REGION

REGION Network 8
   // 旋转到夹紧位置
   // ENO of a box is taken as its EN; it also drops when the box reports an error
   #MC_MoveAbsolute_Instance_5(Axis := "输入轴驱动伺服-1",   // MC_MoveAbsolute
                           Execute := #"Step" = 6,
                           Position := "SERVER_DB".复检参数[2],
                           Velocity := 20.0,
                           Done => #Temp[1]);
   IF #Temp[1] THEN
       #"Step" := 7;
       "产品扶持气缸1进" := TRUE;
       "产品扶持气缸1退" := FALSE;
   END_IF;
END_REGION

REGION Network 9: 下降到接近位置
   // ENO of a box is taken as its EN; it also drops when the box reports an error
   #MC_MoveAbsolute_Instance(Axis := #Axis,   // MC_MoveAbsolute
                           Execute := #"Step" = 7,
                           Position := #接近位置,
                           Velocity := #接近速度,
                           Done => #Temp[2]);
   IF #Temp[2] THEN #"Step" := 8; END_IF;
END_REGION

REGION Network 10: 慢速下降套花键
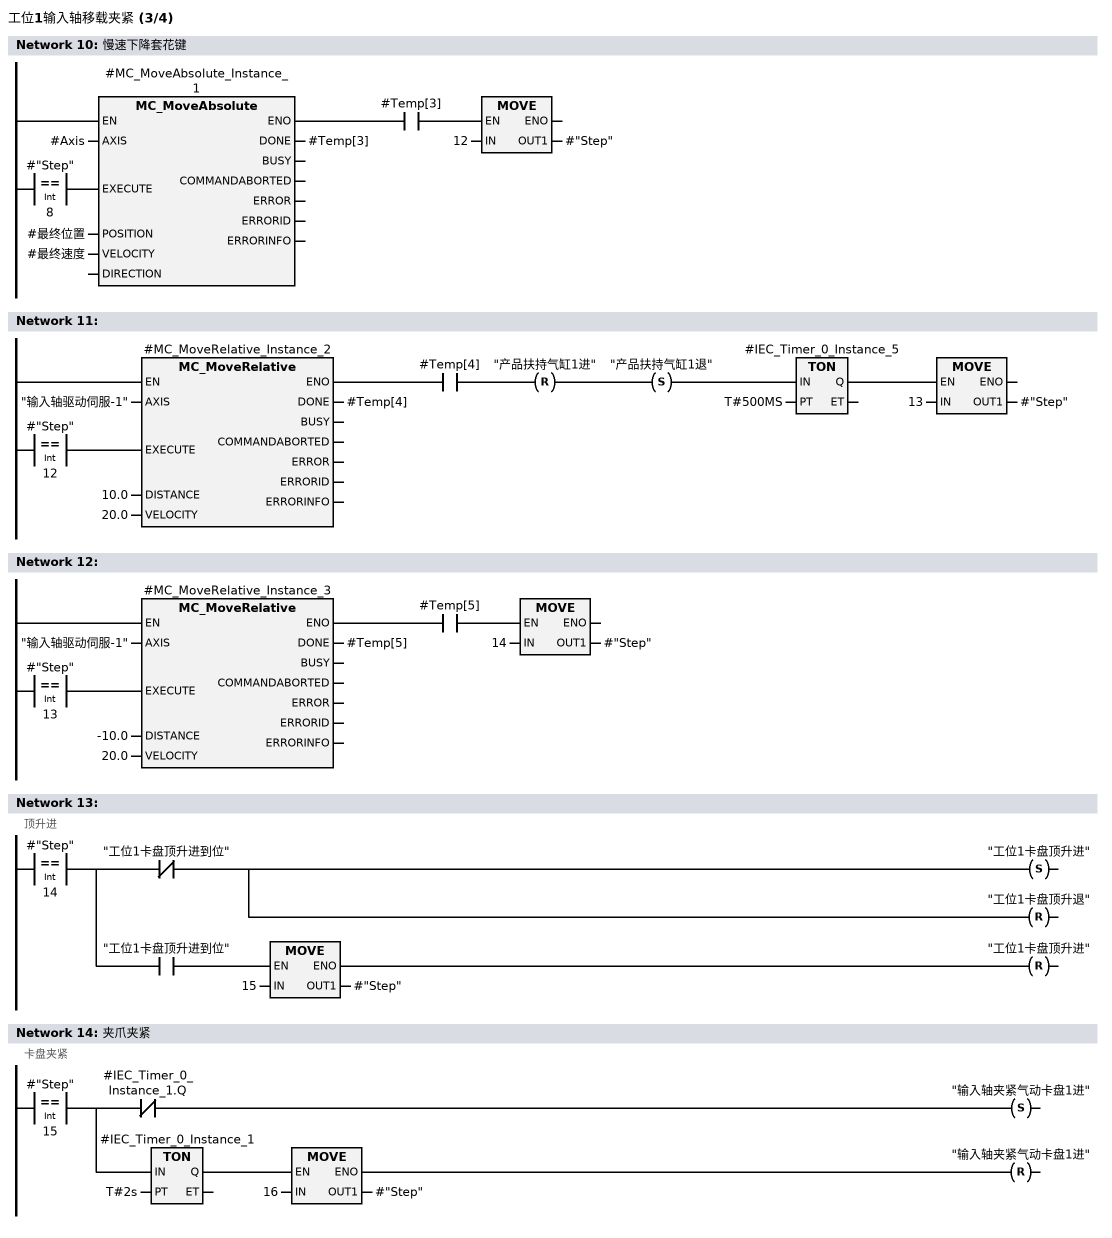
   // ENO of a box is taken as its EN; it also drops when the box reports an error
   #MC_MoveAbsolute_Instance_1(Axis := #Axis,   // MC_MoveAbsolute
                           Execute := #"Step" = 8,
                           Position := #最终位置,
                           Velocity := #最终速度,
                           Done => #Temp[3]);
   IF #Temp[3] THEN #"Step" := 12; END_IF;
END_REGION

REGION Network 11
   // ENO of a box is taken as its EN; it also drops when the box reports an error
   #MC_MoveRelative_Instance_2(Axis := "输入轴驱动伺服-1",   // MC_MoveRelative
                           Execute := #"Step" = 12,
                           Distance := 10.0,
                           Velocity := 20.0,
                           Done => #Temp[4]);
   IF #Temp[4] THEN
       "产品扶持气缸1进" := FALSE;
       "产品扶持气缸1退" := TRUE;
   END_IF;
   #IEC_Timer_0_Instance_5(IN := #Temp[4], PT := T#500MS);   // TON
   IF #IEC_Timer_0_Instance_5.Q THEN #"Step" := 13; END_IF;
END_REGION

REGION Network 12
   // ENO of a box is taken as its EN; it also drops when the box reports an error
   #MC_MoveRelative_Instance_3(Axis := "输入轴驱动伺服-1",   // MC_MoveRelative
                           Execute := #"Step" = 13,
                           Distance := -10.0,
                           Velocity := 20.0,
                           Done => #Temp[5]);
   IF #Temp[5] THEN #"Step" := 14; END_IF;
END_REGION

REGION Network 13
   // 顶升进
   RUNG wire#powerrail
      { S7_Templates := "SrcType := Int" } EQ_Contact(in1 := #"Step", in2 := 14)
      wire#w1
      I_Contact( "工位1卡盘顶升进到位" )
      wire#w2
      S_Coil( "工位1卡盘顶升进" )
   END_RUNG
   RUNG wire#w2
      R_Coil( "工位1卡盘顶升退" )
   END_RUNG
   RUNG wire#w1
      Contact( "工位1卡盘顶升进到位" )
      Move(in := 15, out1 => #"Step")
      R_Coil( "工位1卡盘顶升进" )
   END_RUNG
   // the same network as SCL:
   #_w1 := #"Step" = 14;
   IF #_w1 AND NOT "工位1卡盘顶升进到位" THEN
       "工位1卡盘顶升进" := TRUE;
       "工位1卡盘顶升退" := FALSE;
   END_IF;
   IF #_w1 AND "工位1卡盘顶升进到位" THEN
       #"Step" := 15;
       "工位1卡盘顶升进" := FALSE;
   END_IF;
END_REGION

REGION Network 14: 夹爪夹紧
   // 卡盘夹紧
   #_w1 := #"Step" = 15;
   IF #_w1 AND NOT #IEC_Timer_0_Instance_1.Q THEN "输入轴夹紧气动卡盘1进" := TRUE; END_IF;
   #IEC_Timer_0_Instance_1(IN := #_w1, PT := T#2s);   // TON
   IF #IEC_Timer_0_Instance_1.Q THEN
       #"Step" := 16;
       "输入轴夹紧气动卡盘1进" := FALSE;
   END_IF;
END_REGION

REGION Network 15
   // 顶升退
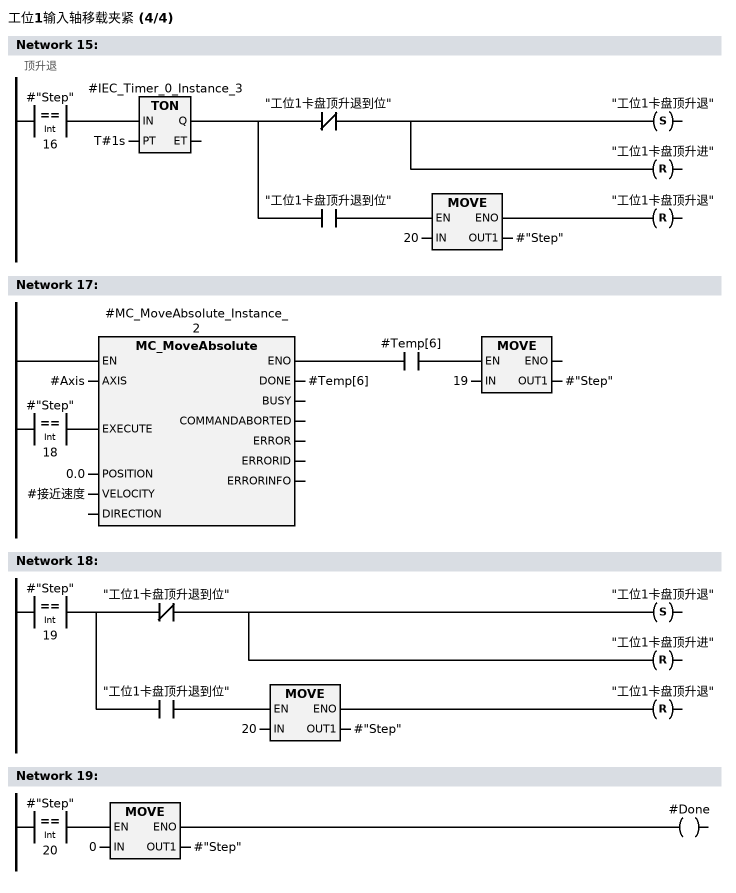
   #IEC_Timer_0_Instance_3(IN := #"Step" = 16, PT := T#1s);   // TON
   IF #IEC_Timer_0_Instance_3.Q AND NOT "工位1卡盘顶升退到位" THEN
       "工位1卡盘顶升退" := TRUE;
       "工位1卡盘顶升进" := FALSE;
   END_IF;
   IF #IEC_Timer_0_Instance_3.Q AND "工位1卡盘顶升退到位" THEN
       #"Step" := 20;
       "工位1卡盘顶升退" := FALSE;
   END_IF;
END_REGION

REGION Network 16: 松开步骤开始
END_REGION

REGION Network 17
   // ENO of a box is taken as its EN; it also drops when the box reports an error
   #MC_MoveAbsolute_Instance_2(Axis := #Axis,   // MC_MoveAbsolute
                           Execute := #"Step" = 18,
                           Position := 0.0,
                           Velocity := #接近速度,
                           Done => #Temp[6]);
   IF #Temp[6] THEN #"Step" := 19; END_IF;
END_REGION

REGION Network 18
   RUNG wire#powerrail
      { S7_Templates := "SrcType := Int" } EQ_Contact(in1 := #"Step", in2 := 19)
      wire#w1
      I_Contact( "工位1卡盘顶升退到位" )
      wire#w2
      S_Coil( "工位1卡盘顶升退" )
   END_RUNG
   RUNG wire#w2
      R_Coil( "工位1卡盘顶升进" )
   END_RUNG
   RUNG wire#w1
      Contact( "工位1卡盘顶升退到位" )
      Move(in := 20, out1 => #"Step")
      R_Coil( "工位1卡盘顶升退" )
   END_RUNG
   // the same network as SCL:
   #_w1 := #"Step" = 19;
   IF #_w1 AND NOT "工位1卡盘顶升退到位" THEN
       "工位1卡盘顶升退" := TRUE;
       "工位1卡盘顶升进" := FALSE;
   END_IF;
   IF #_w1 AND "工位1卡盘顶升退到位" THEN
       #"Step" := 20;
       "工位1卡盘顶升退" := FALSE;
   END_IF;
END_REGION

REGION Network 19
   RUNG wire#powerrail
      { S7_Templates := "SrcType := Int" } EQ_Contact(in1 := #"Step", in2 := 20)
      Move(in := 0, out1 => #"Step")
      Coil( #Done )
   END_RUNG
   // the same network as SCL:
   #_w1 := #"Step" = 20;
   IF #_w1 THEN #"Step" := 0; END_IF;
   #Done := #_w1;
END_REGION
END_FUNCTION_BLOCK

FUNCTION_BLOCK "工位2复检"   // FB13, LAD
{ S7_Optimized_Access := 'TRUE' }
VERSION : 0.1
   VAR_INPUT
      Aix_In : TO_PositioningAxis;
      Excute : Bool;
      Clamp : Bool;
      Test_Speed : Real;
      Status : Byte;
      Stop : Bool;
   END_VAR
   VAR_OUTPUT
      Done : Bool;
   END_VAR
   VAR
      "Step" : Int;
      Test_Velocity : Real;
      Temp : Array[0..7] of Bool;
      MC_Halt_Instance : MC_Halt;
      MC_Halt_Instance_1 : MC_Halt;
      MC_MoveVelocity_Instance : MC_MoveVelocity;
      IEC_Timer_0_Instance : TON_TIME;
      工位2输入轴二次夹紧_Instance : "工位2输入轴二次夹紧";
   END_VAR
   VAR_TEMP   // added for the SCL form of the ladder/FBD networks
      _w1 : Bool;
      _w2 : Bool;
   END_VAR
BEGIN

REGION Network 1
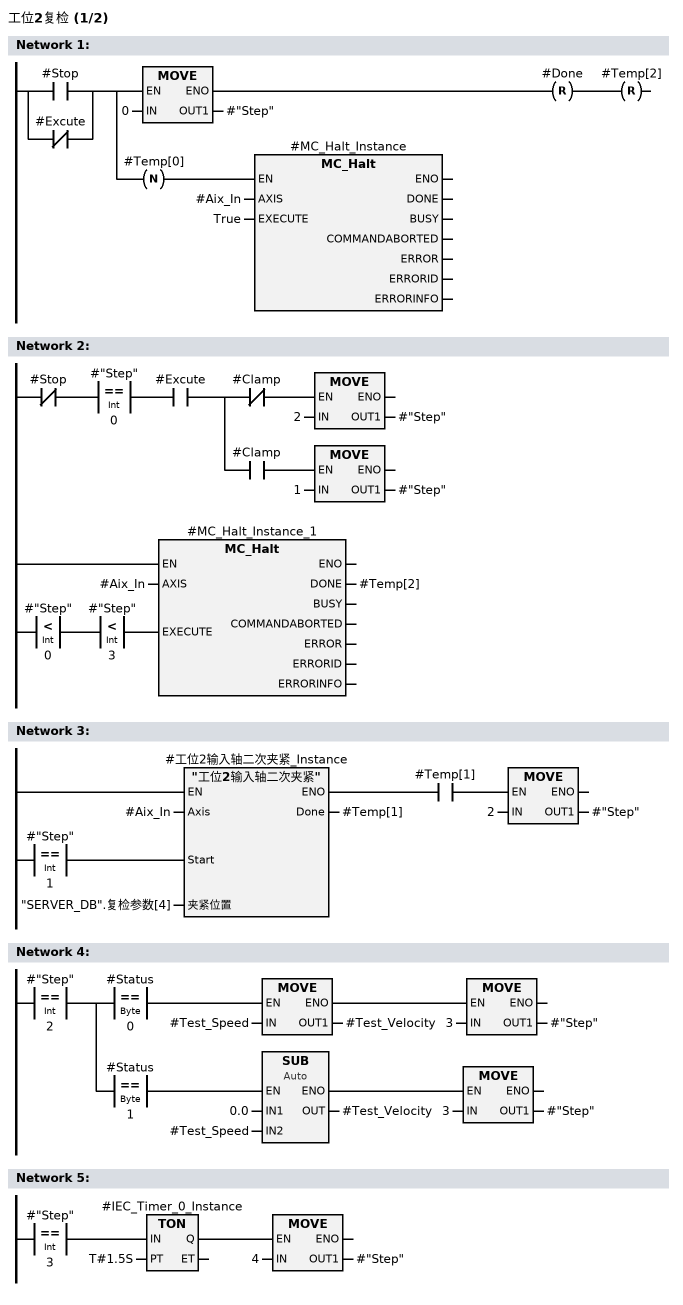
   #_w1 := #Stop OR NOT #Excute;
   IF #_w1 THEN
       #"Step" := 0;
       #Done := FALSE;
       #Temp[2] := FALSE;
   END_IF;
   #_w2 := NOT #_w1 AND #Temp[0];   // falling edge
   #Temp[0] := #_w1;
   IF #_w2 THEN
       #MC_Halt_Instance(Axis := #Aix_In, Execute := True);   // MC_Halt
   END_IF;
END_REGION

REGION Network 2
   #_w1 := NOT #Stop AND (#"Step" = 0) AND #Excute;
   IF #_w1 AND NOT #Clamp THEN #"Step" := 2; END_IF;
   IF #_w1 AND #Clamp THEN #"Step" := 1; END_IF;
   #MC_Halt_Instance_1(Axis := #Aix_In, Execute := (#"Step" < 0) AND (#"Step" < 3), Done => #Temp[2]);   // MC_Halt
END_REGION

REGION Network 3
   RUNG wire#powerrail
      #工位2输入轴二次夹紧_Instance(Start := wire#w1, Axis := #Aix_In, 夹紧位置 := "SERVER_DB".复检参数[4], Done => #Temp[1])
      Contact( #Temp[1] )
      Move(in := 2, out1 => #"Step")
   END_RUNG
   RUNG wire#powerrail
      { S7_Templates := "SrcType := Int" } EQ_Contact(in1 := #"Step", in2 := 1)
   END_RUNG wire#w1
   // the same network as SCL:
   #工位2输入轴二次夹紧_Instance(Axis := #Aix_In,   // "工位2输入轴二次夹紧"
                        Start := #"Step" = 1,
                        夹紧位置 := "SERVER_DB".复检参数[4],
                        Done => #Temp[1],
                        ENO => #_w1);
   IF #_w1 AND #Temp[1] THEN #"Step" := 2; END_IF;
END_REGION

REGION Network 4
   RUNG wire#powerrail
      { S7_Templates := "SrcType := Int" } EQ_Contact(in1 := #"Step", in2 := 2)
      wire#w1
      { S7_Templates := "SrcType := Byte" } EQ_Contact(in1 := #Status, in2 := 0)
      Move(in := #Test_Speed, out1 => #Test_Velocity)
      Move(in := 3, out1 => #"Step")
   END_RUNG
   RUNG wire#w1
      { S7_Templates := "SrcType := Byte" } EQ_Contact(in1 := #Status, in2 := 1)
      Sub(in1 := 0.0, in2 := #Test_Speed, out => #Test_Velocity)
      Move(in := 3, out1 => #"Step")
   END_RUNG
   // the same network as SCL:
   #_w1 := #"Step" = 2;
   IF #_w1 AND (#Status = 0) THEN
       #Test_Velocity := #Test_Speed;
       #"Step" := 3;
   END_IF;
   IF #_w1 AND (#Status = 1) THEN
       #Test_Velocity := 0.0 - #Test_Speed;
       #"Step" := 3;
   END_IF;
END_REGION

REGION Network 5
   #IEC_Timer_0_Instance(IN := #"Step" = 3, PT := T#1.5S);   // TON
   IF #IEC_Timer_0_Instance.Q THEN #"Step" := 4; END_IF;
END_REGION

REGION Network 6
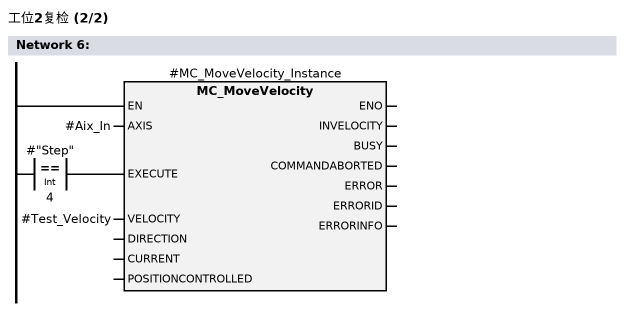
   #MC_MoveVelocity_Instance(Axis := #Aix_In, Execute := #"Step" = 4, Velocity := #Test_Velocity);   // MC_MoveVelocity
END_REGION
END_FUNCTION_BLOCK

FUNCTION_BLOCK "工位2输入轴二次夹紧"   // FB14, LAD
{ S7_Optimized_Access := 'TRUE' }
VERSION : 0.1
   VAR_INPUT
      Axis : TO_PositioningAxis;
      Start : Bool;
      夹紧位置 : Real;
   END_VAR
   VAR_OUTPUT
      Done : Bool;
   END_VAR
   VAR
      "Step" : Int;
      Temp : Array[0..3] of Bool;
      MC_MoveAbsolute_Instance : MC_MoveAbsolute;
      IEC_Timer_0_Instance : TON_TIME;
      IEC_Timer_0_Instance_1 : TON_TIME;
   END_VAR
   VAR_TEMP   // added for the SCL form of the ladder/FBD networks
      _w1 : Bool;
   END_VAR
BEGIN

REGION Network 1
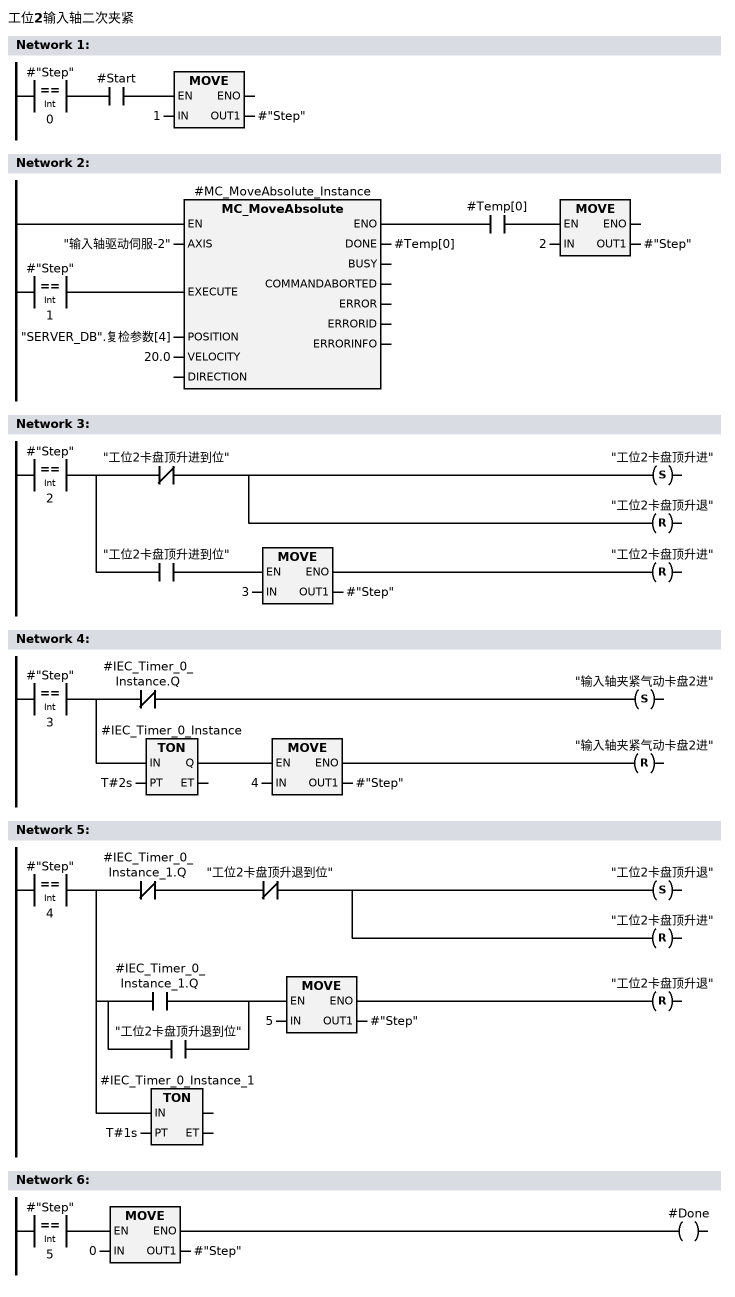
   RUNG wire#powerrail
      { S7_Templates := "SrcType := Int" } EQ_Contact(in1 := #"Step", in2 := 0)
      Contact( #Start )
      Move(in := 1, out1 => #"Step")
   END_RUNG
   // the same network as SCL:
   IF (#"Step" = 0) AND #Start THEN #"Step" := 1; END_IF;
END_REGION

REGION Network 2
   // ENO of a box is taken as its EN; it also drops when the box reports an error
   #MC_MoveAbsolute_Instance(Axis := "输入轴驱动伺服-2",   // MC_MoveAbsolute
                           Execute := #"Step" = 1,
                           Position := "SERVER_DB".复检参数[4],
                           Velocity := 20.0,
                           Done => #Temp[0]);
   IF #Temp[0] THEN #"Step" := 2; END_IF;
END_REGION

REGION Network 3
   RUNG wire#powerrail
      { S7_Templates := "SrcType := Int" } EQ_Contact(in1 := #"Step", in2 := 2)
      wire#w1
      I_Contact( "工位2卡盘顶升进到位" )
      wire#w2
      S_Coil( "工位2卡盘顶升进" )
   END_RUNG
   RUNG wire#w2
      R_Coil( "工位2卡盘顶升退" )
   END_RUNG
   RUNG wire#w1
      Contact( "工位2卡盘顶升进到位" )
      Move(in := 3, out1 => #"Step")
      R_Coil( "工位2卡盘顶升进" )
   END_RUNG
   // the same network as SCL:
   #_w1 := #"Step" = 2;
   IF #_w1 AND NOT "工位2卡盘顶升进到位" THEN
       "工位2卡盘顶升进" := TRUE;
       "工位2卡盘顶升退" := FALSE;
   END_IF;
   IF #_w1 AND "工位2卡盘顶升进到位" THEN
       #"Step" := 3;
       "工位2卡盘顶升进" := FALSE;
   END_IF;
END_REGION

REGION Network 4
   #_w1 := #"Step" = 3;
   IF #_w1 AND NOT #IEC_Timer_0_Instance.Q THEN "输入轴夹紧气动卡盘2进" := TRUE; END_IF;
   #IEC_Timer_0_Instance(IN := #_w1, PT := T#2s);   // TON
   IF #IEC_Timer_0_Instance.Q THEN
       #"Step" := 4;
       "输入轴夹紧气动卡盘2进" := FALSE;
   END_IF;
END_REGION

REGION Network 5
   #_w1 := #"Step" = 4;
   IF #_w1 AND NOT #IEC_Timer_0_Instance_1.Q AND NOT "工位2卡盘顶升退到位" THEN
       "工位2卡盘顶升退" := TRUE;
       "工位2卡盘顶升进" := FALSE;
   END_IF;
   IF #_w1 AND (#IEC_Timer_0_Instance_1.Q OR "工位2卡盘顶升退到位") THEN
       #"Step" := 5;
       "工位2卡盘顶升退" := FALSE;
   END_IF;
   #IEC_Timer_0_Instance_1(IN := #_w1, PT := T#1s);   // TON
END_REGION

REGION Network 6
   RUNG wire#powerrail
      { S7_Templates := "SrcType := Int" } EQ_Contact(in1 := #"Step", in2 := 5)
      Move(in := 0, out1 => #"Step")
      Coil( #Done )
   END_RUNG
   // the same network as SCL:
   #_w1 := #"Step" = 5;
   IF #_w1 THEN #"Step" := 0; END_IF;
   #Done := #_w1;
END_REGION
END_FUNCTION_BLOCK

FUNCTION_BLOCK "工位2输入轴移载夹紧"   // FB15, LAD
{ S7_Optimized_Access := 'TRUE' }
VERSION : 0.1
   VAR_INPUT
      Axis : TO_PositioningAxis;
      接近位置 : Real;
      接近速度 : Real;
      最终位置 : Real;
      最终速度 : Real;
      夹紧 : Bool;
      松开 : Bool;
   END_VAR
   VAR_OUTPUT
      Done : Bool;
   END_VAR
   VAR
      "Step" : Int;
      Temp : Array[0..7] of Bool;
      MC_MoveAbsolute_Instance : MC_MoveAbsolute;
      MC_MoveAbsolute_Instance_1 : MC_MoveAbsolute;
      MC_MoveAbsolute_Instance_2 : MC_MoveAbsolute;
      IEC_Timer_0_Instance : TON_TIME;
      IEC_Timer_0_Instance_1 : TON_TIME;
      MC_MoveAbsolute_Instance_3 : MC_MoveAbsolute;
      MC_MoveAbsolute_Instance_4 : MC_MoveAbsolute;
      MC_MoveAbsolute_Instance_5 : MC_MoveAbsolute;
      IEC_Timer_0_Instance_2 : TON_TIME;
      IEC_Timer_0_Instance_3 : TON_TIME;
      IEC_Timer_0_Instance_4 : TON_TIME;
      MC_MoveRelative_Instance : MC_MoveRelative;
      MC_MoveRelative_Instance_1 : MC_MoveRelative;
   END_VAR
   VAR RETAIN
      IEC_Counter_0_Instance : CTU_INT;
   END_VAR
   VAR
      MC_MoveRelative_Instance_2 : MC_MoveRelative;
      MC_MoveRelative_Instance_3 : MC_MoveRelative;
      IEC_Timer_0_Instance_5 : TON_TIME;
   END_VAR
   VAR_TEMP   // added for the SCL form of the ladder/FBD networks
      _w1 : Bool;
   END_VAR
BEGIN

REGION Network 1
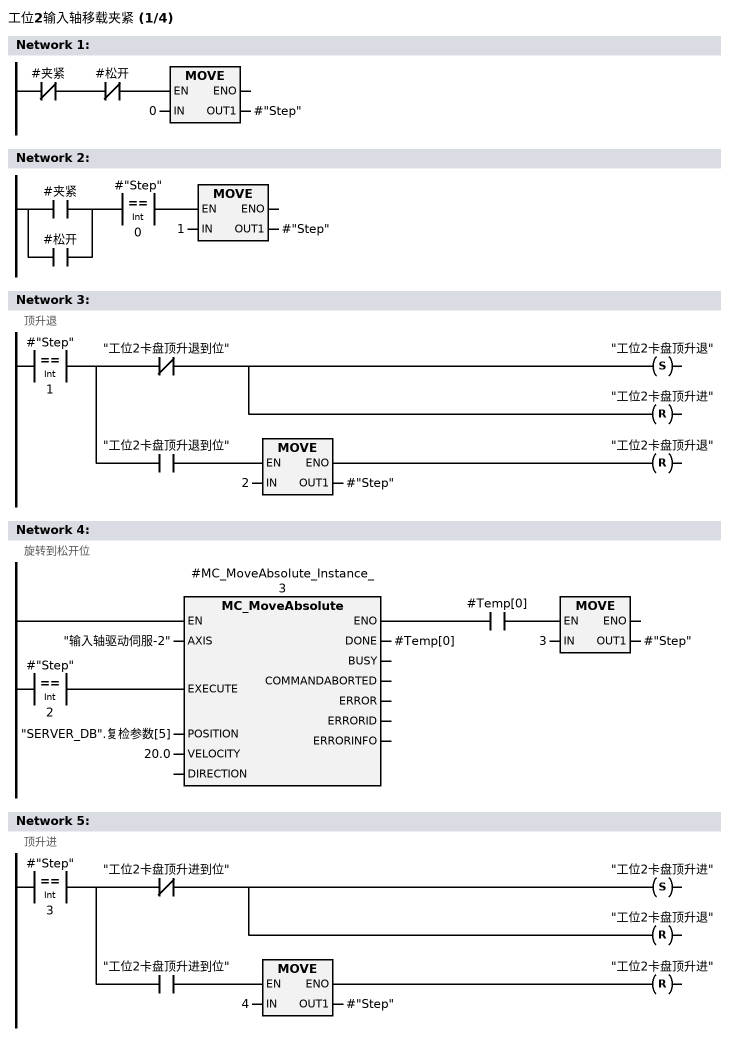
   RUNG wire#powerrail
      I_Contact( #夹紧 )
      I_Contact( #松开 )
      Move(in := 0, out1 => #"Step")
   END_RUNG
   // the same network as SCL:
   IF NOT #夹紧 AND NOT #松开 THEN #"Step" := 0; END_IF;
END_REGION

REGION Network 2
   RUNG wire#powerrail
      Contact( #夹紧 )
      wire#w1
      { S7_Templates := "SrcType := Int" } EQ_Contact(in1 := #"Step", in2 := 0)
      Move(in := 1, out1 => #"Step")
   END_RUNG
   RUNG wire#powerrail
      Contact( #松开 )
   END_RUNG wire#w1
   // the same network as SCL:
   IF (#夹紧 OR #松开) AND (#"Step" = 0) THEN #"Step" := 1; END_IF;
END_REGION

REGION Network 3
   // 顶升退
   RUNG wire#powerrail
      { S7_Templates := "SrcType := Int" } EQ_Contact(in1 := #"Step", in2 := 1)
      wire#w1
      I_Contact( "工位2卡盘顶升退到位" )
      wire#w2
      S_Coil( "工位2卡盘顶升退" )
   END_RUNG
   RUNG wire#w2
      R_Coil( "工位2卡盘顶升进" )
   END_RUNG
   RUNG wire#w1
      Contact( "工位2卡盘顶升退到位" )
      Move(in := 2, out1 => #"Step")
      R_Coil( "工位2卡盘顶升退" )
   END_RUNG
   // the same network as SCL:
   #_w1 := #"Step" = 1;
   IF #_w1 AND NOT "工位2卡盘顶升退到位" THEN
       "工位2卡盘顶升退" := TRUE;
       "工位2卡盘顶升进" := FALSE;
   END_IF;
   IF #_w1 AND "工位2卡盘顶升退到位" THEN
       #"Step" := 2;
       "工位2卡盘顶升退" := FALSE;
   END_IF;
END_REGION

REGION Network 4
   // 旋转到松开位
   // ENO of a box is taken as its EN; it also drops when the box reports an error
   #MC_MoveAbsolute_Instance_3(Axis := "输入轴驱动伺服-2",   // MC_MoveAbsolute
                           Execute := #"Step" = 2,
                           Position := "SERVER_DB".复检参数[5],
                           Velocity := 20.0,
                           Done => #Temp[0]);
   IF #Temp[0] THEN #"Step" := 3; END_IF;
END_REGION

REGION Network 5
   // 顶升进
   RUNG wire#powerrail
      { S7_Templates := "SrcType := Int" } EQ_Contact(in1 := #"Step", in2 := 3)
      wire#w1
      I_Contact( "工位2卡盘顶升进到位" )
      wire#w2
      S_Coil( "工位2卡盘顶升进" )
   END_RUNG
   RUNG wire#w2
      R_Coil( "工位2卡盘顶升退" )
   END_RUNG
   RUNG wire#w1
      Contact( "工位2卡盘顶升进到位" )
      Move(in := 4, out1 => #"Step")
      R_Coil( "工位2卡盘顶升进" )
   END_RUNG
   // the same network as SCL:
   #_w1 := #"Step" = 3;
   IF #_w1 AND NOT "工位2卡盘顶升进到位" THEN
       "工位2卡盘顶升进" := TRUE;
       "工位2卡盘顶升退" := FALSE;
   END_IF;
   IF #_w1 AND "工位2卡盘顶升进到位" THEN
       #"Step" := 4;
       "工位2卡盘顶升进" := FALSE;
   END_IF;
END_REGION

REGION Network 6
   // 卡盘松开
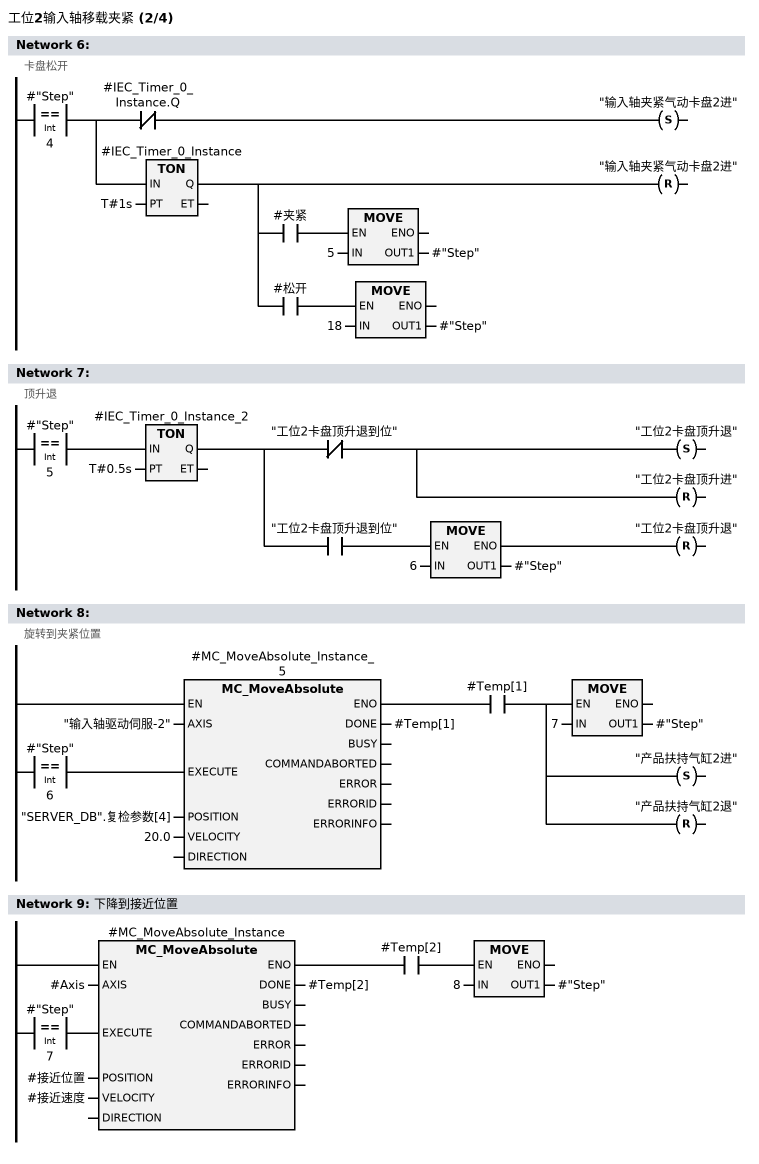
   #_w1 := #"Step" = 4;
   IF #_w1 AND NOT #IEC_Timer_0_Instance.Q THEN "输入轴夹紧气动卡盘2进" := TRUE; END_IF;
   #IEC_Timer_0_Instance(IN := #_w1, PT := T#1s);   // TON
   IF #IEC_Timer_0_Instance.Q THEN "输入轴夹紧气动卡盘2进" := FALSE; END_IF;
   IF #IEC_Timer_0_Instance.Q AND #夹紧 THEN #"Step" := 5; END_IF;
   IF #IEC_Timer_0_Instance.Q AND #松开 THEN #"Step" := 18; END_IF;
END_REGION

REGION Network 7
   // 顶升退
   #IEC_Timer_0_Instance_2(IN := #"Step" = 5, PT := T#0.5s);   // TON
   IF #IEC_Timer_0_Instance_2.Q AND NOT "工位2卡盘顶升退到位" THEN
       "工位2卡盘顶升退" := TRUE;
       "工位2卡盘顶升进" := FALSE;
   END_IF;
   IF #IEC_Timer_0_Instance_2.Q AND "工位2卡盘顶升退到位" THEN
       #"Step" := 6;
       "工位2卡盘顶升退" := FALSE;
   END_IF;
END_REGION

REGION Network 8
   // 旋转到夹紧位置
   // ENO of a box is taken as its EN; it also drops when the box reports an error
   #MC_MoveAbsolute_Instance_5(Axis := "输入轴驱动伺服-2",   // MC_MoveAbsolute
                           Execute := #"Step" = 6,
                           Position := "SERVER_DB".复检参数[4],
                           Velocity := 20.0,
                           Done => #Temp[1]);
   IF #Temp[1] THEN
       #"Step" := 7;
       "产品扶持气缸2进" := TRUE;
       "产品扶持气缸2退" := FALSE;
   END_IF;
END_REGION

REGION Network 9: 下降到接近位置
   // ENO of a box is taken as its EN; it also drops when the box reports an error
   #MC_MoveAbsolute_Instance(Axis := #Axis,   // MC_MoveAbsolute
                           Execute := #"Step" = 7,
                           Position := #接近位置,
                           Velocity := #接近速度,
                           Done => #Temp[2]);
   IF #Temp[2] THEN #"Step" := 8; END_IF;
END_REGION

REGION Network 10: 慢速下降套花键
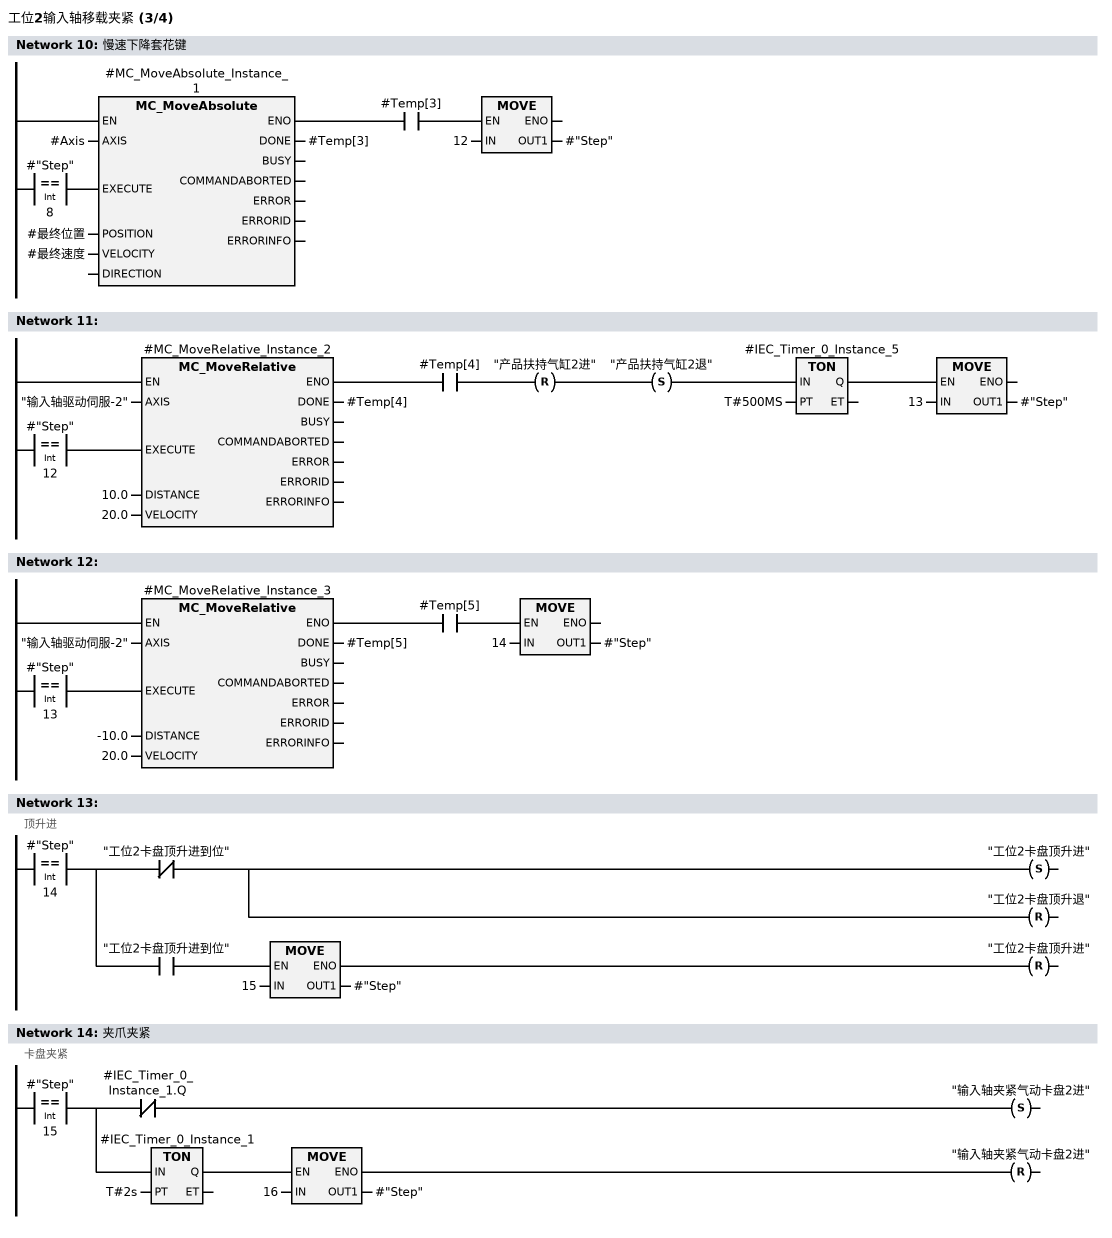
   // ENO of a box is taken as its EN; it also drops when the box reports an error
   #MC_MoveAbsolute_Instance_1(Axis := #Axis,   // MC_MoveAbsolute
                           Execute := #"Step" = 8,
                           Position := #最终位置,
                           Velocity := #最终速度,
                           Done => #Temp[3]);
   IF #Temp[3] THEN #"Step" := 12; END_IF;
END_REGION

REGION Network 11
   // ENO of a box is taken as its EN; it also drops when the box reports an error
   #MC_MoveRelative_Instance_2(Axis := "输入轴驱动伺服-2",   // MC_MoveRelative
                           Execute := #"Step" = 12,
                           Distance := 10.0,
                           Velocity := 20.0,
                           Done => #Temp[4]);
   IF #Temp[4] THEN
       "产品扶持气缸2进" := FALSE;
       "产品扶持气缸2退" := TRUE;
   END_IF;
   #IEC_Timer_0_Instance_5(IN := #Temp[4], PT := T#500MS);   // TON
   IF #IEC_Timer_0_Instance_5.Q THEN #"Step" := 13; END_IF;
END_REGION

REGION Network 12
   // ENO of a box is taken as its EN; it also drops when the box reports an error
   #MC_MoveRelative_Instance_3(Axis := "输入轴驱动伺服-2",   // MC_MoveRelative
                           Execute := #"Step" = 13,
                           Distance := -10.0,
                           Velocity := 20.0,
                           Done => #Temp[5]);
   IF #Temp[5] THEN #"Step" := 14; END_IF;
END_REGION

REGION Network 13
   // 顶升进
   RUNG wire#powerrail
      { S7_Templates := "SrcType := Int" } EQ_Contact(in1 := #"Step", in2 := 14)
      wire#w1
      I_Contact( "工位2卡盘顶升进到位" )
      wire#w2
      S_Coil( "工位2卡盘顶升进" )
   END_RUNG
   RUNG wire#w2
      R_Coil( "工位2卡盘顶升退" )
   END_RUNG
   RUNG wire#w1
      Contact( "工位2卡盘顶升进到位" )
      Move(in := 15, out1 => #"Step")
      R_Coil( "工位2卡盘顶升进" )
   END_RUNG
   // the same network as SCL:
   #_w1 := #"Step" = 14;
   IF #_w1 AND NOT "工位2卡盘顶升进到位" THEN
       "工位2卡盘顶升进" := TRUE;
       "工位2卡盘顶升退" := FALSE;
   END_IF;
   IF #_w1 AND "工位2卡盘顶升进到位" THEN
       #"Step" := 15;
       "工位2卡盘顶升进" := FALSE;
   END_IF;
END_REGION

REGION Network 14: 夹爪夹紧
   // 卡盘夹紧
   #_w1 := #"Step" = 15;
   IF #_w1 AND NOT #IEC_Timer_0_Instance_1.Q THEN "输入轴夹紧气动卡盘2进" := TRUE; END_IF;
   #IEC_Timer_0_Instance_1(IN := #_w1, PT := T#2s);   // TON
   IF #IEC_Timer_0_Instance_1.Q THEN
       #"Step" := 16;
       "输入轴夹紧气动卡盘2进" := FALSE;
   END_IF;
END_REGION

REGION Network 15
   // 顶升退
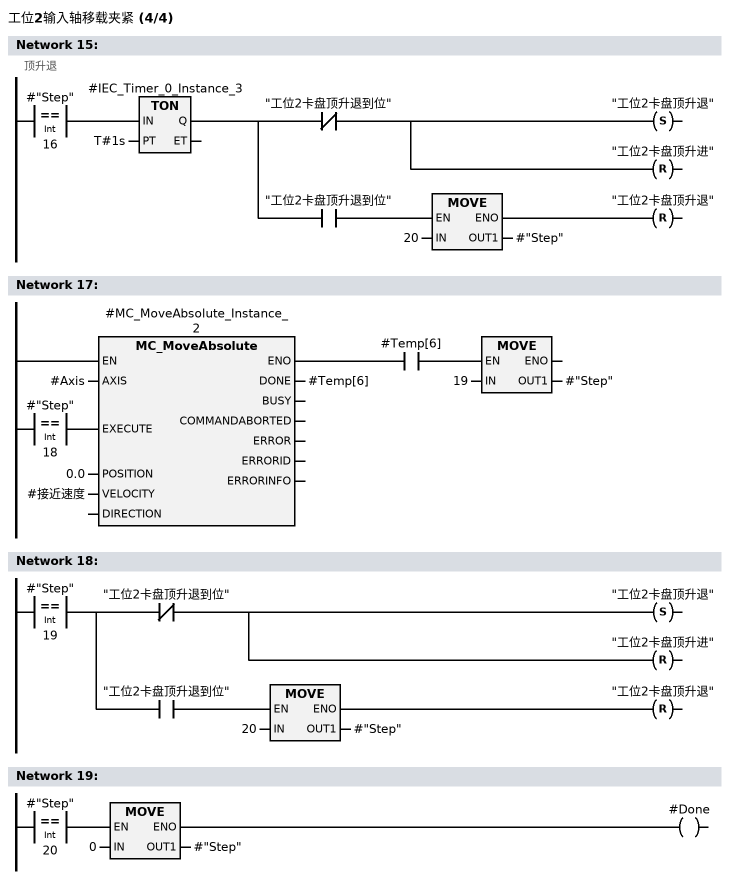
   #IEC_Timer_0_Instance_3(IN := #"Step" = 16, PT := T#1s);   // TON
   IF #IEC_Timer_0_Instance_3.Q AND NOT "工位2卡盘顶升退到位" THEN
       "工位2卡盘顶升退" := TRUE;
       "工位2卡盘顶升进" := FALSE;
   END_IF;
   IF #IEC_Timer_0_Instance_3.Q AND "工位2卡盘顶升退到位" THEN
       #"Step" := 20;
       "工位2卡盘顶升退" := FALSE;
   END_IF;
END_REGION

REGION Network 16: 松开步骤开始
END_REGION

REGION Network 17
   // ENO of a box is taken as its EN; it also drops when the box reports an error
   #MC_MoveAbsolute_Instance_2(Axis := #Axis,   // MC_MoveAbsolute
                           Execute := #"Step" = 18,
                           Position := 0.0,
                           Velocity := #接近速度,
                           Done => #Temp[6]);
   IF #Temp[6] THEN #"Step" := 19; END_IF;
END_REGION

REGION Network 18
   RUNG wire#powerrail
      { S7_Templates := "SrcType := Int" } EQ_Contact(in1 := #"Step", in2 := 19)
      wire#w1
      I_Contact( "工位2卡盘顶升退到位" )
      wire#w2
      S_Coil( "工位2卡盘顶升退" )
   END_RUNG
   RUNG wire#w2
      R_Coil( "工位2卡盘顶升进" )
   END_RUNG
   RUNG wire#w1
      Contact( "工位2卡盘顶升退到位" )
      Move(in := 20, out1 => #"Step")
      R_Coil( "工位2卡盘顶升退" )
   END_RUNG
   // the same network as SCL:
   #_w1 := #"Step" = 19;
   IF #_w1 AND NOT "工位2卡盘顶升退到位" THEN
       "工位2卡盘顶升退" := TRUE;
       "工位2卡盘顶升进" := FALSE;
   END_IF;
   IF #_w1 AND "工位2卡盘顶升退到位" THEN
       #"Step" := 20;
       "工位2卡盘顶升退" := FALSE;
   END_IF;
END_REGION

REGION Network 19
   RUNG wire#powerrail
      { S7_Templates := "SrcType := Int" } EQ_Contact(in1 := #"Step", in2 := 20)
      Move(in := 0, out1 => #"Step")
      Coil( #Done )
   END_RUNG
   // the same network as SCL:
   #_w1 := #"Step" = 20;
   IF #_w1 THEN #"Step" := 0; END_IF;
   #Done := #_w1;
END_REGION
END_FUNCTION_BLOCK

FUNCTION "Analog To Project amount" : Void   // FC1, LAD
{ S7_Optimized_Access := 'TRUE' }
VERSION : 0.1
   VAR_INPUT
      Analog : Int;
      Min_Value : Real;
      Max_Value : Real;
   END_VAR
   VAR_OUTPUT
      Project_amount : Real;
   END_VAR
   VAR_TEMP
      Temp_Value : Real;
   END_VAR
BEGIN

REGION Network 1
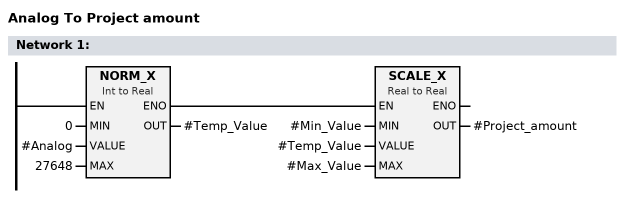
   RUNG wire#powerrail
      { S7_Templates := "[SrcType := Int, DestType := Real]" } Normalize(min := 0, value := #Analog, max := 27648, out => #Temp_Value)
      { S7_Templates := "[SrcType := Real, DestType := Real]" } Scale(min := #Min_Value, value := #Temp_Value, max := #Max_Value, out => #Project_amount)
   END_RUNG
   // the same network as SCL:
   #Temp_Value := NORM_X(MIN := 0, VALUE := #Analog, MAX := 27648);
   #Project_amount := SCALE_X(MIN := #Min_Value, VALUE := #Temp_Value, MAX := #Max_Value);
END_REGION
END_FUNCTION

FUNCTION "encoder" : Void   // FC2, LAD
{ S7_Optimized_Access := 'TRUE' }
VERSION : 0.1
   VAR_INPUT
      encoder : DInt;
   END_VAR
   VAR_OUTPUT
      angle : Real;
   END_VAR
   VAR_TEMP
      Temp_Value : DInt;
      Temp_Value2 : DInt;
   END_VAR
BEGIN

REGION Network 1
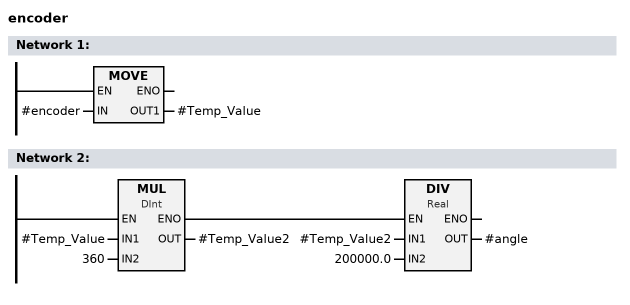
   RUNG wire#powerrail
      Move(in := #encoder, out1 => #Temp_Value)
   END_RUNG
   // the same network as SCL:
   #Temp_Value := #encoder;
END_REGION

REGION Network 2
   RUNG wire#powerrail
      { S7_Templates := "SrcType := DInt" } Mul(in1 := #Temp_Value, in2 := 360, out => #Temp_Value2)
      { S7_Templates := "SrcType := Real" } Div(in1 := #Temp_Value2, in2 := 200000.0, out => #angle)
   END_RUNG
   // the same network as SCL:
   #Temp_Value2 := #Temp_Value * 360;
   #angle := #Temp_Value2 / 200000.0;
END_REGION
END_FUNCTION

ORGANIZATION_BLOCK "Main"   // OB1, LAD, ProgramCycle
TITLE = "Main Program Sweep (Cycle)"
{ S7_Optimized_Access := 'TRUE' }
VERSION : 0.1
   VAR_INPUT
      Initial_Call : Bool;   // Initial call of this OB
      Remanence : Bool;   // =True, if remanent data are available
   END_VAR
   VAR_TEMP   // added for the SCL form of the ladder/FBD networks
      _w1 : Bool;
      _w2 : Bool;
   END_VAR
BEGIN

REGION Network 1
